C03643=1208.967,92.723,-48.603,-178.715,5.757,148.635
C03644=1208.971,92.474,-48.585,-178.717,5.756,148.636
C03645=1208.975,92.224,-48.566,-178.719,5.755,148.636
C03646=1208.980,91.975,-48.548,-178.723,5.754,148.637
C03647=1208.985,91.726,-48.530,-178.725,5.753,148.637
C03648=1208.990,91.477,-48.512,-178.727,5.752,148.638
C03649=1208.996,91.227,-48.494,-178.731,5.751,148.639
C03650=1209.000,90.977,-48.475,-178.733,5.750,148.639
C03651=1209.005,90.728,-48.457,-178.735,5.749,148.640
C03652=1209.010,90.479,-48.440,-178.737,5.748,148.640
C03653=1209.015,90.230,-48.422,-178.741,5.747,148.641
C03654=1209.020,89.981,-48.404,-178.743,5.746,148.642
C03655=1209.025,89.732,-48.386,-178.745,5.746,148.642
C03656=1209.029,89.482,-48.367,-178.748,5.745,148.643
C03657=1209.034,89.232,-48.349,-178.751,5.744,148.643
C03658=1209.039,88.983,-48.331,-178.753,5.743,148.644
C03659=1209.044,88.734,-48.313,-178.756,5.742,148.644
C03660=1209.049,88.485,-48.295,-178.758,5.741,148.645
C03661=1209.054,88.236,-48.277,-178.761,5.740,148.645
C03662=1209.059,87.987,-48.259,-178.764,5.739,148.646
C03663=1209.064,87.736,-48.240,-178.766,5.738,148.646
C03664=1209.068,87.487,-48.222,-178.769,5.738,148.647
C03665=1209.073,87.238,-48.204,-178.771,5.736,148.648
C03666=1209.078,86.989,-48.186,-178.774,5.735,148.648
C03667=1209.083,86.740,-48.168,-178.777,5.735,148.649
C03668=1209.088,86.491,-48.151,-178.779,5.734,148.649
C03669=1209.093,86.241,-48.133,-178.782,5.732,148.650
C03670=1209.097,85.993,-48.115,-178.785,5.732,148.651
C03671=1209.102,85.743,-48.097,-178.787,5.731,148.651
C03672=1209.107,85.493,-48.080,-178.789,5.730,148.652
C03673=1209.112,85.244,-48.062,-178.793,5.729,148.652
C03674=1209.117,84.994,-48.044,-178.795,5.728,148.653
C03675=1209.121,84.745,-48.026,-178.797,5.727,148.653
C03676=1209.126,84.496,-48.008,-178.799,5.726,148.654
C03677=1209.131,84.247,-47.990,-178.803,5.725,148.654
C03678=1209.137,83.997,-47.972,-178.805,5.725,148.655
C03679=1209.141,83.748,-47.954,-178.807,5.724,148.655
C03680=1209.146,83.499,-47.936,-178.810,5.723,148.656
C03681=1209.151,83.250,-47.918,-178.813,5.722,148.657
C03682=1209.156,83.000,-47.900,-178.815,5.721,148.657
C03683=1209.161,82.751,-47.883,-178.818,5.720,148.658
C03684=1209.166,82.501,-47.865,-178.821,5.720,148.659
C03685=1209.170,82.253,-47.848,-178.823,5.719,148.659
C03686=1209.175,82.003,-47.829,-178.826,5.717,148.660
C03687=1209.180,81.753,-47.812,-178.829,5.717,148.660
C03688=1209.186,81.485,-47.793,-178.831,5.716,148.661
C03689=1209.191,81.217,-47.774,-178.834,5.714,148.661
C03690=1209.196,80.948,-47.755,-178.837,5.714,148.662
C03691=1209.201,80.680,-47.736,-178.839,5.713,148.663
C03692=1209.206,80.431,-47.718,-178.842,5.712,148.663
C03693=1209.211,80.181,-47.700,-178.844,5.711,148.664
C03694=1209.216,79.932,-47.682,-178.847,5.710,148.664
C03695=1209.220,79.683,-47.665,-178.850,5.710,148.665
C03696=1209.226,79.433,-47.648,-178.852,5.709,148.665
C03697=1209.231,79.184,-47.630,-178.855,5.707,148.666
C03698=1209.236,78.935,-47.612,-178.858,5.707,148.667
C03699=1209.241,78.685,-47.595,-178.860,5.706,148.667
C03700=1209.245,78.436,-47.577,-178.862,5.705,148.668
C03701=1209.250,78.186,-47.560,-178.865,5.705,148.669
C03702=1209.255,77.937,-47.542,-178.868,5.703,148.669
C03703=1209.260,77.688,-47.524,-178.870,5.702,148.670
C03704=1209.264,77.439,-47.507,-178.873,5.702,148.670
C03705=1209.269,77.189,-47.489,-178.875,5.701,148.671
C03706=1209.275,76.940,-47.472,-178.878,5.700,148.671
C03707=1209.279,76.690,-47.454,-178.881,5.699,148.672
C03708=1209.284,76.441,-47.437,-178.883,5.698,148.672
C03709=1209.289,76.192,-47.419,-178.886,5.698,148.673
C03710=1209.294,75.942,-47.402,-178.888,5.697,148.674
C03711=1209.300,75.693,-47.385,-178.891,5.696,148.674
C03712=1209.304,75.444,-47.368,-178.894,5.695,148.675
C03713=1209.309,75.195,-47.350,-178.896,5.694,148.675
C03714=1209.314,74.945,-47.333,-178.898,5.693,148.676
C03715=1209.318,74.696,-47.315,-178.901,5.693,148.677
C03716=1209.324,74.446,-47.298,-178.904,5.692,148.677
C03717=1209.329,74.197,-47.280,-178.906,5.691,148.678
C03718=1209.334,73.947,-47.263,-178.909,5.690,148.678
C03719=1209.338,73.699,-47.245,-178.912,5.689,148.679
C03720=1209.343,73.449,-47.228,-178.914,5.688,148.679
C03721=1209.348,73.200,-47.210,-178.916,5.688,148.680
C03722=1209.353,72.950,-47.193,-178.919,5.687,148.681
C03723=1209.358,72.701,-47.177,-178.922,5.685,148.681
C03724=1209.362,72.452,-47.159,-178.924,5.685,148.682
C03725=1209.368,72.202,-47.142,-178.927,5.684,148.682
C03726=1209.373,71.953,-47.124,-178.930,5.684,148.683
C03727=1209.377,71.704,-47.107,-178.932,5.683,148.684
C03728=1209.382,71.454,-47.090,-178.934,5.682,148.684
C03729=1209.387,71.205,-47.072,-178.937,5.682,148.685
C03730=1209.392,70.956,-47.056,-178.940,5.680,148.685
C03731=1209.398,70.706,-47.038,-178.942,5.679,148.686
C03732=1209.402,70.457,-47.021,-178.945,5.679,148.687
C03733=1209.407,70.207,-47.004,-178.947,5.678,148.687
C03734=1209.412,69.958,-46.987,-178.950,5.677,148.688
C03735=1209.416,69.709,-46.969,-178.952,5.677,148.688
C03736=1209.422,69.459,-46.952,-178.956,5.675,148.689
C03737=1209.427,69.210,-46.936,-178.958,5.674,148.689
C03738=1209.432,68.961,-46.918,-178.960,5.674,148.690
C03739=1209.436,68.712,-46.901,-178.963,5.673,148.691
C03740=1209.441,68.462,-46.884,-178.965,5.672,148.691
C03741=1209.446,68.212,-46.867,-178.968,5.672,148.692
C03742=1209.451,67.963,-46.849,-178.970,5.671,148.693
C03743=1209.456,67.714,-46.833,-178.973,5.669,148.693
C03744=1209.461,67.465,-46.815,-178.976,5.669,148.694
C03745=1209.465,67.215,-46.799,-178.978,5.668,148.694
C03746=1209.470,66.966,-46.781,-178.981,5.668,148.695
C03747=1209.475,66.716,-46.764,-178.983,5.667,148.695
C03748=1209.481,66.467,-46.747,-178.986,5.666,148.696
C03749=1209.485,66.218,-46.731,-178.988,5.666,148.697
C03750=1209.490,65.968,-46.713,-178.991,5.664,148.697
C03751=1209.495,65.719,-46.697,-178.994,5.663,148.698
C03752=1209.500,65.470,-46.679,-178.996,5.663,148.698
C03753=1209.505,65.221,-46.662,-178.999,5.662,148.699
C03754=1209.510,64.971,-46.645,-179.001,5.661,148.700
C03755=1209.514,64.721,-46.628,-179.004,5.661,148.700
C03756=1209.520,64.471,-46.611,-179.007,5.660,148.701
C03757=1209.525,64.223,-46.595,-179.009,5.659,148.701
C03758=1209.529,63.973,-46.578,-179.012,5.658,148.702
C03759=1209.534,63.723,-46.561,-179.014,5.657,148.703
C03760=1209.539,63.475,-46.544,-179.017,5.657,148.703
C03761=1209.544,63.225,-46.527,-179.019,5.656,148.704
C03762=1209.549,62.976,-46.510,-179.022,5.655,148.704
C03763=1209.554,62.726,-46.493,-179.025,5.655,148.705
C03764=1209.559,62.477,-46.476,-179.027,5.654,148.706
C03765=1209.564,62.228,-46.460,-179.029,5.653,148.706
C03766=1209.569,61.978,-46.442,-179.033,5.652,148.707
C03767=1209.573,61.729,-46.426,-179.035,5.651,148.707
C03768=1209.579,61.480,-46.409,-179.037,5.651,148.708
C03769=1209.584,61.230,-46.392,-179.040,5.650,148.709
C03770=1209.588,60.981,-46.376,-179.043,5.649,148.709
C03771=1209.594,60.732,-46.359,-179.045,5.649,148.710
C03772=1209.599,60.482,-46.342,-179.047,5.648,148.710
C03773=1209.603,60.233,-46.325,-179.050,5.647,148.711
C03774=1209.609,59.983,-46.308,-179.053,5.647,148.712
C03775=1209.613,59.734,-46.292,-179.055,5.646,148.712
C03776=1209.618,59.484,-46.275,-179.058,5.645,148.713
C03777=1209.623,59.235,-46.258,-179.061,5.644,148.713
C03778=1209.628,58.986,-46.241,-179.063,5.643,148.714
C03779=1209.633,58.736,-46.226,-179.066,5.643,148.715
C03780=1209.637,58.486,-46.209,-179.068,5.642,148.715
C03781=1209.643,58.237,-46.192,-179.071,5.641,148.716
C03782=1209.648,57.988,-46.175,-179.073,5.641,148.717
C03783=1209.653,57.739,-46.159,-179.076,5.640,148.717
C03784=1209.658,57.489,-46.142,-179.078,5.639,148.718
C03785=1209.662,57.240,-46.125,-179.081,5.639,148.718
C03786=1209.667,56.991,-46.109,-179.084,5.638,148.719
C03787=1209.672,56.741,-46.092,-179.087,5.637,148.720
C03788=1209.677,56.491,-46.076,-179.089,5.636,148.720
C03789=1209.683,56.242,-46.059,-179.091,5.636,148.721
C03790=1209.687,55.993,-46.043,-179.094,5.635,148.721
C03791=1209.692,55.743,-46.026,-179.097,5.634,148.722
C03792=1209.698,55.474,-46.008,-179.099,5.634,148.723
C03793=1209.703,55.207,-45.991,-179.102,5.633,148.723
C03794=1209.708,54.938,-45.972,-179.105,5.632,148.724
C03795=1209.713,54.670,-45.955,-179.107,5.631,148.724
C03796=1209.719,54.420,-45.938,-179.110,5.630,148.725
C03797=1209.724,54.171,-45.922,-179.112,5.630,148.726
C03798=1209.728,53.921,-45.905,-179.115,5.629,148.726
C03799=1209.733,53.671,-45.889,-179.118,5.629,148.727
C03800=1209.738,53.423,-45.873,-179.120,5.628,148.728
C03801=1209.743,53.173,-45.856,-179.123,5.627,148.728
C03802=1209.749,52.923,-45.840,-179.125,5.627,148.729
C03803=1209.753,52.674,-45.823,-179.128,5.626,148.730
C03804=1209.758,52.425,-45.807,-179.130,5.625,148.730
C03805=1209.763,52.176,-45.790,-179.133,5.624,148.731
C03806=1209.767,51.926,-45.774,-179.136,5.623,148.731
C03807=1209.772,51.677,-45.758,-179.138,5.623,148.732
C03808=1209.778,51.427,-45.741,-179.141,5.622,148.732
C03809=1209.783,51.178,-45.725,-179.143,5.621,148.733
C03810=1209.788,50.928,-45.709,-179.146,5.621,148.734
C03811=1209.793,50.679,-45.692,-179.148,5.620,148.734
C03812=1209.797,50.429,-45.676,-179.151,5.619,148.735
C03813=1209.802,50.180,-45.660,-179.153,5.619,148.736
C03814=1209.807,49.930,-45.644,-179.156,5.618,148.736
C03815=1209.812,49.682,-45.628,-179.159,5.618,148.737
C03816=1209.817,49.432,-45.611,-179.161,5.617,148.738
C03817=1209.822,49.183,-45.596,-179.163,5.616,148.738
C03818=1209.827,48.933,-45.579,-179.166,5.616,148.739
C03819=1209.833,48.683,-45.563,-179.169,5.615,148.739
C03820=1209.837,48.434,-45.546,-179.171,5.615,148.740
C03821=1209.843,48.185,-45.530,-179.173,5.614,148.740
C03822=1209.847,47.935,-45.514,-179.176,5.613,148.741
C03823=1209.852,47.686,-45.498,-179.179,5.613,148.742
C03824=1209.857,47.436,-45.482,-179.181,5.612,148.743
C03825=1209.862,47.187,-45.465,-179.185,5.611,148.743
C03826=1209.867,46.937,-45.449,-179.187,5.610,148.744
C03827=1209.872,46.689,-45.433,-179.189,5.609,148.744
C03828=1209.877,46.438,-45.417,-179.192,5.609,148.745
C03829=1209.882,46.190,-45.401,-179.195,5.608,148.746
C03830=1209.887,45.940,-45.385,-179.197,5.608,148.746
C03831=1209.892,45.691,-45.368,-179.199,5.607,148.747
C03832=1209.896,45.441,-45.353,-179.202,5.606,148.747
C03833=1209.902,45.191,-45.337,-179.205,5.606,148.748
C03834=1209.906,44.942,-45.320,-179.207,5.605,148.749
C03835=1209.912,44.692,-45.305,-179.210,5.605,148.749
C03836=1209.916,44.443,-45.288,-179.212,5.604,148.750
C03837=1209.922,44.193,-45.272,-179.215,5.603,148.751
C03838=1209.927,43.945,-45.256,-179.217,5.603,148.751
C03839=1209.931,43.695,-45.241,-179.220,5.602,148.752
C03840=1209.936,43.445,-45.225,-179.222,5.601,148.752
C03841=1209.941,43.196,-45.209,-179.225,5.601,148.753
C03842=1209.946,42.947,-45.193,-179.227,5.600,148.754
C03843=1209.951,42.696,-45.177,-179.230,5.600,148.754
C03844=1209.956,42.448,-45.161,-179.233,5.599,148.755
C03845=1209.961,42.198,-45.145,-179.235,5.598,148.755
C03846=1209.966,41.949,-45.128,-179.237,5.598,148.756
C03847=1209.971,41.699,-45.113,-179.240,5.597,148.757
C03848=1209.976,41.449,-45.097,-179.243,5.597,148.757
C03849=1209.981,41.200,-45.081,-179.245,5.596,148.758
C03850=1209.986,40.951,-45.066,-179.248,5.595,148.759
C03851=1209.990,40.701,-45.050,-179.250,5.595,148.759
C03852=1209.996,40.452,-45.034,-179.253,5.594,148.760
C03853=1210.001,40.203,-45.018,-179.255,5.594,148.761
C03854=1210.006,39.953,-45.002,-179.258,5.593,148.761
C03855=1210.011,39.704,-44.986,-179.260,5.592,148.762
C03856=1210.016,39.454,-44.970,-179.263,5.592,148.762
C03857=1210.020,39.205,-44.955,-179.266,5.591,148.763
C03858=1210.026,38.956,-44.939,-179.268,5.590,148.764
C03859=1210.030,38.706,-44.923,-179.271,5.590,148.764
C03860=1210.036,38.456,-44.907,-179.273,5.589,148.765
C03861=1210.041,38.207,-44.891,-179.276,5.588,148.766
C03862=1210.046,37.957,-44.875,-179.278,5.588,148.766
C03863=1210.050,37.708,-44.860,-179.281,5.587,148.767
C03864=1210.056,37.459,-44.845,-179.284,5.587,148.768
C03865=1210.060,37.209,-44.829,-179.286,5.586,148.768
C03866=1210.066,36.960,-44.812,-179.288,5.585,148.769
C03867=1210.071,36.710,-44.797,-179.291,5.585,148.769
C03868=1210.075,36.461,-44.781,-179.294,5.584,148.770
C03869=1210.080,36.211,-44.766,-179.296,5.584,148.771
C03870=1210.086,35.962,-44.750,-179.299,5.583,148.771
C03871=1210.091,35.712,-44.735,-179.301,5.582,148.772
C03872=1210.095,35.463,-44.719,-179.304,5.582,148.773
C03873=1210.101,35.213,-44.704,-179.306,5.581,148.773
C03874=1210.106,34.965,-44.687,-179.309,5.581,148.774
C03875=1210.110,34.714,-44.671,-179.312,5.580,148.775
C03876=1210.115,34.465,-44.656,-179.314,5.580,148.775
C03877=1210.120,34.216,-44.641,-179.316,5.579,148.776
C03878=1210.125,33.966,-44.625,-179.319,5.578,148.776
C03879=1210.130,33.717,-44.610,-179.322,5.578,148.777
C03880=1210.135,33.467,-44.594,-179.324,5.577,148.778
C03881=1210.141,33.218,-44.579,-179.327,5.577,148.778
C03882=1210.145,32.968,-44.563,-179.330,5.576,148.779
C03883=1210.150,32.719,-44.548,-179.332,5.575,148.779
C03884=1210.155,32.469,-44.532,-179.334,5.575,148.780
C03885=1210.161,32.220,-44.517,-179.336,5.575,148.781
C03886=1210.165,31.970,-44.501,-179.339,5.574,148.782
C03887=1210.170,31.721,-44.486,-179.342,5.574,148.782
C03888=1210.175,31.472,-44.471,-179.344,5.573,148.783
C03889=1210.180,31.222,-44.455,-179.347,5.573,148.783
C03890=1210.185,30.972,-44.439,-179.349,5.572,148.784
C03891=1210.190,30.723,-44.424,-179.352,5.571,148.785
C03892=1210.195,30.474,-44.408,-179.355,5.571,148.785
C03893=1210.201,30.224,-44.393,-179.357,5.570,148.786
C03894=1210.205,29.975,-44.378,-179.360,5.570,148.787
C03895=1210.210,29.725,-44.362,-179.362,5.569,148.787
C03896=1210.216,29.456,-44.346,-179.365,5.568,148.788
C03897=1210.221,29.188,-44.329,-179.367,5.568,148.789
C03898=1210.226,28.919,-44.312,-179.370,5.568,148.789
C03899=1210.232,28.650,-44.296,-179.373,5.567,148.790
C03900=1210.237,28.401,-44.281,-179.375,5.566,148.791
C03901=1210.242,28.152,-44.265,-179.378,5.566,148.791
C03902=1210.246,27.902,-44.250,-179.380,5.565,148.792
C03903=1210.252,27.652,-44.234,-179.383,5.565,148.793
C03904=1210.256,27.403,-44.219,-179.386,5.564,148.793
C03905=1210.262,27.153,-44.205,-179.388,5.564,148.794
C03906=1210.267,26.904,-44.190,-179.391,5.563,148.794
C03907=1210.272,26.655,-44.174,-179.393,5.562,148.795
C03908=1210.277,26.405,-44.158,-179.396,5.562,148.796
C03909=1210.281,26.156,-44.143,-179.398,5.561,148.796
C03910=1210.287,25.906,-44.128,-179.401,5.561,148.797
C03911=1210.292,25.657,-44.113,-179.404,5.560,148.798
C03912=1210.297,25.407,-44.098,-179.406,5.560,148.798
C03913=1210.302,25.158,-44.083,-179.409,5.559,148.799
C03914=1210.307,24.908,-44.067,-179.411,5.559,148.800
C03915=1210.311,24.658,-44.052,-179.413,5.559,148.800
C03916=1210.317,24.409,-44.037,-179.416,5.558,148.801
C03917=1210.322,24.160,-44.022,-179.419,5.557,148.802
C03918=1210.327,23.910,-44.006,-179.421,5.557,148.802
C03919=1210.332,23.661,-43.992,-179.423,5.556,148.803
C03920=1210.337,23.412,-43.977,-179.426,5.556,148.803
C03921=1210.342,23.162,-43.961,-179.429,5.555,148.804
C03922=1210.346,22.912,-43.947,-179.431,5.555,148.805
C03923=1210.352,22.662,-43.931,-179.434,5.554,148.805
C03924=1210.356,22.413,-43.916,-179.437,5.553,148.806
C03925=1210.362,22.164,-43.900,-179.439,5.553,148.807
C03926=1210.367,21.914,-43.886,-179.441,5.552,148.807
C03927=1210.372,21.665,-43.871,-179.443,5.552,148.808
C03928=1210.377,21.416,-43.856,-179.446,5.552,148.809
C03929=1210.382,21.166,-43.841,-179.449,5.551,148.809
C03930=1210.387,20.917,-43.826,-179.451,5.551,148.810
C03931=1210.392,20.667,-43.811,-179.454,5.550,148.811
C03932=1210.397,20.417,-43.796,-179.457,5.550,148.811
C03933=1210.401,20.168,-43.781,-179.459,5.549,148.812
C03934=1210.406,19.918,-43.766,-179.462,5.548,148.813
C03935=1210.412,19.669,-43.751,-179.464,5.548,148.813
C03936=1210.417,19.419,-43.736,-179.467,5.547,148.814
C03937=1210.422,19.169,-43.721,-179.469,5.547,148.815
C03938=1210.427,18.920,-43.706,-179.472,5.547,148.815
C03939=1210.432,18.671,-43.692,-179.474,5.547,148.816
C03940=1210.437,18.421,-43.676,-179.476,5.546,148.816
C03941=1210.442,18.171,-43.662,-179.479,5.545,148.817
C03942=1210.447,17.922,-43.647,-179.482,5.545,148.818
C03943=1210.452,17.672,-43.632,-179.484,5.544,148.818
C03944=1210.457,17.423,-43.617,-179.487,5.544,148.819
C03945=1210.462,17.174,-43.603,-179.490,5.543,148.820
C03946=1210.467,16.924,-43.587,-179.492,5.543,148.820
C03947=1210.472,16.674,-43.573,-179.494,5.542,148.821
C03948=1210.477,16.425,-43.558,-179.496,5.542,148.822
C03949=1210.482,16.176,-43.543,-179.499,5.541,148.822
C03950=1210.487,15.926,-43.528,-179.502,5.541,148.823
C03951=1210.492,15.677,-43.514,-179.504,5.540,148.824
C03952=1210.497,15.427,-43.499,-179.507,5.540,148.824
C03953=1210.503,15.177,-43.484,-179.510,5.539,148.825
C03954=1210.507,14.928,-43.469,-179.512,5.539,148.826
C03955=1210.512,14.679,-43.454,-179.515,5.538,148.826
C03956=1210.517,14.430,-43.439,-179.517,5.538,148.827
C03957=1210.523,14.180,-43.425,-179.519,5.538,148.828
C03958=1210.528,13.930,-43.410,-179.522,5.537,148.828
C03959=1210.532,13.681,-43.395,-179.525,5.537,148.829
C03960=1210.537,13.431,-43.381,-179.527,5.536,148.830
C03961=1210.542,13.182,-43.365,-179.530,5.536,148.830
C03962=1210.547,12.932,-43.351,-179.532,5.535,148.831
C03963=1210.552,12.682,-43.337,-179.535,5.534,148.831
C03964=1210.557,12.433,-43.322,-179.537,5.535,148.832
C03965=1210.562,12.183,-43.308,-179.539,5.534,148.833
C03966=1210.568,11.933,-43.293,-179.542,5.534,148.833
C03967=1210.572,11.684,-43.278,-179.545,5.533,148.834
C03968=1210.577,11.435,-43.263,-179.547,5.532,148.835
C03969=1210.582,11.185,-43.249,-179.550,5.532,148.836
C03970=1210.588,10.936,-43.235,-179.552,5.531,148.836
C03971=1210.593,10.686,-43.220,-179.555,5.531,148.837
C03972=1210.598,10.437,-43.205,-179.557,5.531,148.837
C03973=1210.603,10.188,-43.190,-179.559,5.530,148.838
C03974=1210.608,9.938,-43.176,-179.562,5.530,148.839
C03975=1210.613,9.688,-43.162,-179.565,5.529,148.839
C03976=1210.618,9.439,-43.148,-179.567,5.529,148.840
C03977=1210.623,9.189,-43.132,-179.570,5.528,148.841
C03978=1210.628,8.939,-43.118,-179.573,5.528,148.841
C03979=1210.633,8.690,-43.103,-179.574,5.528,148.842
C03980=1210.638,8.440,-43.089,-179.577,5.527,148.843
C03981=1210.643,8.192,-43.075,-179.580,5.527,148.843
C03982=1210.648,7.942,-43.060,-179.582,5.526,148.844
C03983=1210.653,7.692,-43.046,-179.585,5.526,148.845
C03984=1210.658,7.442,-43.032,-179.588,5.525,148.845
C03985=1210.663,7.193,-43.017,-179.590,5.525,148.846
C03986=1210.668,6.943,-43.002,-179.592,5.525,148.847
C03987=1210.673,6.694,-42.988,-179.594,5.524,148.847
C03988=1210.678,6.444,-42.973,-179.597,5.524,148.848
C03989=1210.684,6.195,-42.959,-179.600,5.523,148.849
C03990=1210.689,5.945,-42.945,-179.602,5.523,148.849
C03991=1210.694,5.695,-42.931,-179.605,5.522,148.850
C03992=1210.698,5.446,-42.916,-179.607,5.522,148.851
C03993=1210.703,5.197,-42.902,-179.610,5.522,148.851
C03994=1210.708,4.947,-42.887,-179.612,5.521,148.852
C03995=1210.713,4.697,-42.873,-179.615,5.521,148.853
C03996=1210.719,4.448,-42.859,-179.617,5.520,148.853
C03997=1210.724,4.199,-42.845,-179.620,5.519,148.854
C03998=1210.729,3.949,-42.831,-179.623,5.519,148.855
C03999=1210.734,3.699,-42.816,-179.625,5.519,148.855
C04000=1210.739,3.430,-42.801,-179.627,5.519,148.856
C04001=1210.744,3.161,-42.786,-179.630,5.518,148.857
C04002=1210.750,2.893,-42.770,-179.633,5.518,148.857
C04003=1210.756,2.623,-42.755,-179.636,5.518,148.858
C04004=1210.761,2.373,-42.740,-179.638,5.517,148.859
C04005=1210.766,2.124,-42.726,-179.641,5.516,148.859
C04006=1210.771,1.874,-42.712,-179.643,5.516,148.860
C04007=1210.776,1.625,-42.698,-179.646,5.515,148.861
C04008=1210.781,1.376,-42.684,-179.648,5.516,148.861
C04009=1210.786,1.126,-42.670,-179.651,5.515,148.862
C04010=1210.791,0.876,-42.656,-179.653,5.514,148.863
C04011=1210.796,0.626,-42.641,-179.656,5.514,148.863
C04012=1210.801,0.377,-42.627,-179.659,5.513,148.864
C04013=1210.806,0.128,-42.613,-179.661,5.513,148.865
C04014=1210.811,-0.122,-42.599,-179.663,5.513,148.865
C04015=1210.816,-0.372,-42.585,-179.665,5.512,148.866
C04016=1210.822,-0.621,-42.571,-179.668,5.512,148.867
C04017=1210.827,-0.870,-42.556,-179.671,5.511,148.867
C04018=1210.832,-1.120,-42.542,-179.673,5.511,148.868
C04019=1210.836,-1.370,-42.528,-179.675,5.511,148.869
C04020=1210.842,-1.619,-42.514,-179.678,5.511,148.869
C04021=1210.846,-1.868,-42.500,-179.681,5.510,148.870
C04022=1210.851,-2.118,-42.486,-179.683,5.510,148.871
C04023=1210.856,-2.368,-42.472,-179.686,5.509,148.871
C04024=1210.862,-2.617,-42.458,-179.688,5.509,148.872
C04025=1210.867,-2.867,-42.444,-179.690,5.509,148.873
C04026=1210.872,-3.117,-42.430,-179.693,5.508,148.873
C04027=1210.877,-3.366,-42.416,-179.696,5.508,148.874
C04028=1210.882,-3.615,-42.402,-179.698,5.507,148.875
C04029=1210.887,-3.865,-42.388,-179.700,5.507,148.875
C04030=1210.892,-4.115,-42.374,-179.703,5.507,148.876
C04031=1210.897,-4.364,-42.361,-179.706,5.506,148.877
C04032=1210.902,-4.614,-42.346,-179.708,5.506,148.877
C04033=1210.907,-4.864,-42.332,-179.711,5.505,148.878
C04034=1210.913,-5.113,-42.318,-179.713,5.505,148.879
C04035=1210.917,-5.362,-42.304,-179.715,5.505,148.879
C04036=1210.922,-5.612,-42.290,-179.718,5.504,148.880
C04037=1210.927,-5.862,-42.277,-179.721,5.504,148.881
C04038=1210.933,-6.111,-42.263,-179.723,5.503,148.881
C04039=1210.938,-6.361,-42.248,-179.725,5.504,148.882
C04040=1210.942,-6.610,-42.235,-179.728,5.503,148.883
C04041=1210.948,-6.860,-42.222,-179.731,5.503,148.883
C04042=1210.953,-7.110,-42.207,-179.733,5.502,148.884
C04043=1210.958,-7.359,-42.193,-179.735,5.501,148.885
C04044=1210.963,-7.608,-42.180,-179.737,5.502,148.885
C04045=1210.968,-7.858,-42.166,-179.740,5.501,148.886
C04046=1210.973,-8.108,-42.152,-179.743,5.501,148.887
C04047=1210.978,-8.357,-42.138,-179.745,5.500,148.887
C04048=1210.983,-8.607,-42.125,-179.748,5.500,148.888
C04049=1210.989,-8.856,-42.111,-179.750,5.500,148.889
C04050=1210.994,-9.106,-42.097,-179.753,5.499,148.889
C04051=1210.999,-9.356,-42.083,-179.755,5.499,148.890
C04052=1211.004,-9.605,-42.070,-179.758,5.498,148.891
C04053=1211.009,-9.854,-42.056,-179.760,5.498,148.891
C04054=1211.014,-10.105,-42.042,-179.762,5.498,148.892
C04055=1211.019,-10.353,-42.029,-179.765,5.497,148.893
C04056=1211.024,-10.603,-42.014,-179.768,5.497,148.893
C04057=1211.029,-10.854,-42.001,-179.770,5.496,148.894
C04058=1211.034,-11.102,-41.988,-179.772,5.497,148.895
C04059=1211.039,-11.352,-41.973,-179.775,5.496,148.895
C04060=1211.044,-11.602,-41.960,-179.778,5.496,148.896
C04061=1211.049,-11.851,-41.946,-179.780,5.495,148.897
C04062=1211.054,-12.101,-41.933,-179.782,5.496,148.898
C04063=1211.060,-12.350,-41.919,-179.785,5.495,148.898
C04064=1211.064,-12.600,-41.906,-179.787,5.494,148.899
C04065=1211.070,-12.849,-41.892,-179.790,5.494,148.899
C04066=1211.075,-13.099,-41.878,-179.793,5.493,148.900
C04067=1211.080,-13.348,-41.865,-179.795,5.494,148.901
C04068=1211.085,-13.598,-41.851,-179.797,5.493,148.901
C04069=1211.090,-13.848,-41.837,-179.800,5.493,148.902
C04070=1211.095,-14.097,-41.824,-179.803,5.492,148.903
C04071=1211.100,-14.347,-41.811,-179.805,5.492,148.904
C04072=1211.105,-14.596,-41.797,-179.807,5.492,148.904
C04073=1211.110,-14.846,-41.784,-179.810,5.491,148.905
C04074=1211.116,-15.095,-41.770,-179.813,5.491,148.906
C04075=1211.120,-15.345,-41.757,-179.814,5.491,148.906
C04076=1211.126,-15.594,-41.743,-179.817,5.490,148.907
C04077=1211.130,-15.845,-41.730,-179.820,5.490,148.907
C04078=1211.136,-16.094,-41.716,-179.822,5.489,148.908
C04079=1211.141,-16.344,-41.702,-179.824,5.490,148.909
C04080=1211.145,-16.593,-41.689,-179.827,5.489,148.910
C04081=1211.151,-16.843,-41.676,-179.830,5.489,148.910
C04082=1211.156,-17.093,-41.663,-179.832,5.488,148.911
C04083=1211.161,-17.342,-41.649,-179.834,5.489,148.912
C04084=1211.166,-17.592,-41.636,-179.837,5.488,148.912
C04085=1211.171,-17.841,-41.622,-179.840,5.488,148.913
C04086=1211.176,-18.091,-41.609,-179.842,5.487,148.914
C04087=1211.182,-18.341,-41.596,-179.844,5.487,148.914
C04088=1211.186,-18.590,-41.582,-179.847,5.487,148.915
C04089=1211.192,-18.840,-41.569,-179.849,5.486,148.916
C04090=1211.197,-19.089,-41.554,-179.852,5.486,148.916
C04091=1211.202,-19.339,-41.542,-179.854,5.486,148.917
C04092=1211.207,-19.589,-41.528,-179.857,5.485,148.918
C04093=1211.212,-19.838,-41.515,-179.859,5.485,148.918
C04094=1211.218,-20.087,-41.502,-179.862,5.484,148.919
C04095=1211.222,-20.337,-41.489,-179.864,5.485,148.920
C04096=1211.227,-20.586,-41.475,-179.867,5.484,148.920
C04097=1211.232,-20.836,-41.462,-179.869,5.484,148.921
C04098=1211.237,-21.086,-41.449,-179.872,5.483,148.922
C04099=1211.242,-21.335,-41.435,-179.874,5.483,148.922
C04100=1211.248,-21.585,-41.422,-179.876,5.483,148.923
C04101=1211.253,-21.835,-41.409,-179.879,5.482,148.924
C04102=1211.258,-22.084,-41.396,-179.881,5.483,148.924
C04103=1211.263,-22.334,-41.382,-179.884,5.482,148.925
C04104=1211.268,-22.603,-41.369,-179.886,5.482,148.926
C04105=1211.274,-22.873,-41.354,-179.889,5.481,148.926
C04106=1211.280,-23.143,-41.339,-179.892,5.481,148.927
C04107=1211.285,-23.412,-41.326,-179.895,5.481,148.928
C04108=1211.290,-23.661,-41.312,-179.897,5.481,148.929
C04109=1211.295,-23.911,-41.299,-179.899,5.480,148.929
C04110=1211.300,-24.161,-41.286,-179.902,5.479,148.930
C04111=1211.306,-24.410,-41.273,-179.904,5.479,148.931
C04112=1211.310,-24.660,-41.260,-179.906,5.479,148.931
C04113=1211.316,-24.909,-41.246,-179.909,5.479,148.932
C04114=1211.321,-25.159,-41.234,-179.912,5.478,148.933
C04115=1211.325,-25.409,-41.221,-179.914,5.479,148.933
C04116=1211.331,-25.658,-41.207,-179.917,5.478,148.934
C04117=1211.336,-25.908,-41.194,-179.919,5.478,148.935
C04118=1211.341,-26.158,-41.182,-179.922,5.477,148.936
C04119=1211.346,-26.407,-41.168,-179.924,5.478,148.936
C04120=1211.351,-26.657,-41.155,-179.927,5.477,148.937
C04121=1211.356,-26.906,-41.142,-179.929,5.476,148.937
C04122=1211.362,-27.156,-41.129,-179.931,5.477,148.938
C04123=1211.367,-27.406,-41.116,-179.933,5.476,148.939
C04124=1211.372,-27.655,-41.104,-179.936,5.476,148.939
C04125=1211.377,-27.905,-41.090,-179.939,5.475,148.940
C04126=1211.382,-28.155,-41.077,-179.941,5.475,148.941
C04127=1211.387,-28.404,-41.065,-179.944,5.475,148.942
C04128=1211.392,-28.654,-41.051,-179.946,5.474,148.942
C04129=1211.397,-28.903,-41.038,-179.948,5.475,148.943
C04130=1211.402,-29.152,-41.025,-179.951,5.474,148.944
C04131=1211.407,-29.402,-41.012,-179.954,5.474,148.944
C04132=1211.413,-29.652,-40.999,-179.956,5.473,148.945
C04133=1211.418,-29.901,-40.987,-179.958,5.473,148.946
C04134=1211.422,-30.151,-40.974,-179.961,5.473,148.946
C04135=1211.428,-30.401,-40.960,-179.963,5.472,148.947
C04136=1211.433,-30.650,-40.948,-179.965,5.473,148.948
C04137=1211.438,-30.900,-40.935,-179.968,5.472,148.948
C04138=1211.443,-31.149,-40.922,-179.971,5.472,148.949
C04139=1211.449,-31.399,-40.909,-179.973,5.472,148.950
C04140=1211.453,-31.649,-40.896,-179.975,5.472,148.950
C04141=1211.459,-31.898,-40.884,-179.978,5.471,148.951
C04142=1211.464,-32.148,-40.871,-179.981,5.471,148.952
C04143=1211.468,-32.398,-40.858,-179.983,5.471,148.952
C04144=1211.474,-32.647,-40.845,-179.985,5.470,148.953
C04145=1211.479,-32.897,-40.832,-179.988,5.470,148.954
C04146=1211.484,-33.146,-40.820,-179.990,5.470,148.954
C04147=1211.489,-33.396,-40.807,-179.992,5.469,148.955
C04148=1211.495,-33.646,-40.793,-179.995,5.469,148.956
C04149=1211.500,-33.896,-40.782,-179.997,5.469,148.956
C04150=1211.505,-34.146,-40.769,-180.000,5.469,148.957
C04151=1211.510,-34.395,-40.756,179.998,5.468,148.958
C04152=1211.515,-34.644,-40.743,179.996,5.469,148.959
C04153=1211.520,-34.894,-40.731,179.993,5.468,148.959
C04154=1211.525,-35.144,-40.717,179.990,5.468,148.960
C04155=1211.530,-35.393,-40.705,179.988,5.467,148.961
C04156=1211.536,-35.643,-40.692,179.985,5.468,148.961
C04157=1211.541,-35.892,-40.679,179.983,5.467,148.962
C04158=1211.545,-36.142,-40.667,179.981,5.466,148.963
C04159=1211.551,-36.392,-40.655,179.979,5.467,148.963
C04160=1211.556,-36.641,-40.641,179.976,5.466,148.964
C04161=1211.562,-36.891,-40.629,179.973,5.466,148.965
C04162=1211.567,-37.140,-40.616,179.971,5.466,148.965
C04163=1211.571,-37.390,-40.603,179.968,5.466,148.966
C04164=1211.577,-37.640,-40.591,179.966,5.465,148.967
C04165=1211.582,-37.889,-40.579,179.964,5.465,148.967
C04166=1211.587,-38.139,-40.566,179.961,5.465,148.968
C04167=1211.591,-38.389,-40.553,179.958,5.464,148.969
C04168=1211.597,-38.638,-40.541,179.957,5.464,148.969
C04169=1211.603,-38.888,-40.528,179.954,5.464,148.970
C04170=1211.608,-39.138,-40.515,179.951,5.463,148.971
C04171=1211.613,-39.387,-40.503,179.949,5.464,148.971
C04172=1211.617,-39.637,-40.490,179.947,5.463,148.972
C04173=1211.623,-39.887,-40.478,179.944,5.463,148.973
C04174=1211.628,-40.136,-40.465,179.942,5.463,148.973
C04175=1211.633,-40.385,-40.453,179.939,5.463,148.974
C04176=1211.639,-40.635,-40.441,179.937,5.462,148.975
C04177=1211.643,-40.885,-40.428,179.935,5.463,148.976
C04178=1211.648,-41.135,-40.415,179.932,5.462,148.976
C04179=1211.653,-41.384,-40.403,179.929,5.462,148.977
C04180=1211.659,-41.634,-40.391,179.928,5.462,148.977
C04181=1211.664,-41.883,-40.378,179.925,5.461,148.978
C04182=1211.669,-42.133,-40.366,179.922,5.461,148.979
C04183=1211.674,-42.383,-40.353,179.920,5.461,148.980
C04184=1211.679,-42.633,-40.341,179.918,5.461,148.980
C04185=1211.684,-42.882,-40.328,179.915,5.460,148.981
C04186=1211.690,-43.132,-40.316,179.913,5.460,148.982
C04187=1211.695,-43.381,-40.304,179.910,5.460,148.982
C04188=1211.700,-43.630,-40.291,179.908,5.459,148.983
C04189=1211.705,-43.880,-40.279,179.905,5.460,148.984
C04190=1211.710,-44.130,-40.266,179.903,5.459,148.984
C04191=1211.715,-44.380,-40.254,179.900,5.459,148.985
C04192=1211.720,-44.630,-40.242,179.899,5.459,148.986
C04193=1211.725,-44.879,-40.229,179.896,5.458,148.986
C04194=1211.731,-45.129,-40.217,179.893,5.458,148.987
C04195=1211.736,-45.378,-40.205,179.891,5.458,148.988
C04196=1211.741,-45.628,-40.193,179.888,5.458,148.988
C04197=1211.747,-45.877,-40.180,179.886,5.458,148.989
C04198=1211.751,-46.128,-40.168,179.884,5.458,148.990
C04199=1211.756,-46.377,-40.155,179.881,5.457,148.991
C04200=1211.762,-46.627,-40.143,179.879,5.458,148.991
C04201=1211.766,-46.876,-40.131,179.876,5.457,148.992
C04202=1211.771,-47.126,-40.119,179.874,5.457,148.993
C04203=1211.777,-47.376,-40.107,179.872,5.457,148.993
C04204=1211.782,-47.625,-40.094,179.869,5.456,148.994
C04205=1211.787,-47.875,-40.082,179.867,5.456,148.995
C04206=1211.793,-48.124,-40.070,179.865,5.456,148.995
C04207=1211.798,-48.374,-40.058,179.862,5.455,148.996
C04208=1211.803,-48.645,-40.045,179.859,5.455,148.997
C04209=1211.808,-48.914,-40.031,179.857,5.455,148.997
C04210=1211.814,-49.184,-40.019,179.854,5.455,148.998
C04211=1211.820,-49.455,-40.005,179.851,5.455,148.999
C04212=1211.825,-49.704,-39.993,179.849,5.454,149.000
C04213=1211.830,-49.953,-39.981,179.847,5.455,149.000
C04214=1211.835,-50.203,-39.969,179.844,5.454,149.001
C04215=1211.841,-50.453,-39.957,179.842,5.453,149.002
C04216=1211.846,-50.702,-39.944,179.840,5.454,149.002
C04217=1211.851,-50.952,-39.932,179.837,5.453,149.003
C04218=1211.856,-51.202,-39.921,179.835,5.454,149.004
C04219=1211.861,-51.451,-39.908,179.832,5.453,149.004
C04220=1211.866,-51.701,-39.897,179.830,5.453,149.005
C04221=1211.871,-51.950,-39.884,179.828,5.453,149.006
C04222=1211.877,-52.200,-39.872,179.825,5.453,149.006
C04223=1211.882,-52.450,-39.860,179.822,5.452,149.007
C04224=1211.887,-52.699,-39.848,179.821,5.452,149.008
C04225=1211.892,-52.949,-39.836,179.818,5.452,149.008
C04226=1211.898,-53.199,-39.824,179.816,5.452,149.009
C04227=1211.903,-53.448,-39.812,179.813,5.451,149.010
C04228=1211.907,-53.698,-39.800,179.811,5.451,149.010
C04229=1211.913,-53.948,-39.789,179.808,5.451,149.011
C04230=1211.918,-54.197,-39.776,179.806,5.451,149.012
C04231=1211.923,-54.447,-39.764,179.803,5.450,149.013
C04232=1211.928,-54.697,-39.753,179.801,5.451,149.013
C04233=1211.933,-54.946,-39.740,179.798,5.450,149.014
C04234=1211.939,-55.196,-39.728,179.796,5.451,149.015
C04235=1211.944,-55.446,-39.716,179.794,5.450,149.015
C04236=1211.948,-55.695,-39.704,179.791,5.449,149.016
C04237=1211.954,-55.945,-39.693,179.789,5.450,149.017
C04238=1211.959,-56.195,-39.681,179.787,5.449,149.017
C04239=1211.964,-56.444,-39.669,179.784,5.449,149.018
C04240=1211.969,-56.694,-39.657,179.782,5.449,149.019
C04241=1211.975,-56.944,-39.645,179.779,5.449,149.019
C04242=1211.980,-57.194,-39.633,179.777,5.449,149.020
C04243=1211.985,-57.443,-39.622,179.774,5.449,149.021
C04244=1211.990,-57.693,-39.609,179.772,5.448,149.022
C04245=1211.995,-57.942,-39.597,179.770,5.448,149.022
C04246=1212.000,-58.192,-39.586,179.768,5.448,149.023
C04247=1212.005,-58.442,-39.574,179.765,5.448,149.023
C04248=1212.011,-58.692,-39.562,179.763,5.448,149.024
C04249=1212.015,-58.941,-39.550,179.760,5.447,149.025
C04250=1212.021,-59.191,-39.538,179.758,5.447,149.026
C04251=1212.026,-59.441,-39.526,179.755,5.447,149.026
C04252=1212.031,-59.690,-39.515,179.753,5.447,149.027
C04253=1212.037,-59.940,-39.504,179.751,5.447,149.028
C04254=1212.042,-60.190,-39.492,179.748,5.446,149.028
C04255=1212.047,-60.439,-39.480,179.746,5.446,149.029
C04256=1212.052,-60.689,-39.468,179.744,5.446,149.030
C04257=1212.057,-60.938,-39.457,179.742,5.446,149.030
C04258=1212.062,-61.188,-39.445,179.739,5.446,149.031
C04259=1212.068,-61.438,-39.433,179.736,5.445,149.032
C04260=1212.072,-61.688,-39.421,179.734,5.446,149.032
C04261=1212.078,-61.938,-39.410,179.732,5.445,149.033
C04262=1212.082,-62.187,-39.398,179.729,5.446,149.034
C04263=1212.088,-62.437,-39.387,179.727,5.445,149.034
C04264=1212.094,-62.686,-39.374,179.724,5.445,149.035
C04265=1212.098,-62.935,-39.363,179.723,5.445,149.036
C04266=1212.104,-63.185,-39.351,179.720,5.444,149.036
C04267=1212.108,-63.435,-39.340,179.718,5.445,149.037
C04268=1212.114,-63.685,-39.328,179.715,5.444,149.038
C04269=1212.118,-63.935,-39.317,179.712,5.444,149.038
C04270=1212.124,-64.185,-39.305,179.710,5.444,149.039
C04271=1212.130,-64.434,-39.293,179.708,5.444,149.040
C04272=1212.135,-64.683,-39.282,179.706,5.444,149.041
C04273=1212.140,-64.933,-39.270,179.703,5.444,149.041
C04274=1212.145,-65.183,-39.259,179.701,5.443,149.042
C04275=1212.150,-65.433,-39.247,179.699,5.443,149.042
C04276=1212.155,-65.683,-39.235,179.696,5.443,149.043
C04277=1212.161,-65.932,-39.224,179.694,5.443,149.044
C04278=1212.166,-66.181,-39.213,179.691,5.442,149.045
C04279=1212.171,-66.431,-39.201,179.689,5.442,149.045
C04280=1212.176,-66.681,-39.190,179.686,5.442,149.046
C04281=1212.181,-66.931,-39.178,179.684,5.442,149.047
C04282=1212.186,-67.180,-39.166,179.682,5.442,149.047
C04283=1212.192,-67.430,-39.155,179.680,5.441,149.048
C04284=1212.197,-67.679,-39.144,179.677,5.442,149.049
C04285=1212.202,-67.930,-39.132,179.675,5.441,149.049
C04286=1212.207,-68.180,-39.121,179.672,5.441,149.050
C04287=1212.212,-68.429,-39.109,179.670,5.441,149.051
C04288=1212.218,-68.678,-39.098,179.667,5.441,149.051
C04289=1212.223,-68.928,-39.086,179.665,5.441,149.052
C04290=1212.228,-69.178,-39.075,179.663,5.441,149.053
C04291=1212.233,-69.428,-39.063,179.660,5.440,149.054
C04292=1212.239,-69.677,-39.052,179.658,5.440,149.054
C04293=1212.243,-69.926,-39.041,179.656,5.440,149.055
C04294=1212.249,-70.176,-39.029,179.654,5.440,149.055
C04295=1212.254,-70.427,-39.019,179.651,5.440,149.056
C04296=1212.259,-70.677,-39.007,179.649,5.440,149.057
C04297=1212.264,-70.925,-38.996,179.646,5.440,149.058
C04298=1212.270,-71.175,-38.984,179.643,5.439,149.058
C04299=1212.274,-71.425,-38.973,179.641,5.440,149.059
C04300=1212.279,-71.675,-38.961,179.639,5.439,149.059
C04301=1212.286,-71.925,-38.950,179.637,5.439,149.060
C04302=1212.290,-72.174,-38.939,179.634,5.439,149.061
C04303=1212.296,-72.424,-38.927,179.632,5.439,149.062
C04304=1212.300,-72.674,-38.916,179.630,5.439,149.062
C04305=1212.306,-72.923,-38.905,179.627,5.438,149.063
C04306=1212.311,-73.173,-38.894,179.625,5.438,149.064
C04307=1212.316,-73.423,-38.883,179.622,5.438,149.064
C04308=1212.322,-73.672,-38.871,179.620,5.438,149.065
C04309=1212.327,-73.922,-38.860,179.618,5.438,149.066
C04310=1212.332,-74.172,-38.849,179.616,5.438,149.066
C04311=1212.337,-74.422,-38.837,179.613,5.437,149.067
C04312=1212.343,-74.692,-38.826,179.611,5.437,149.068
C04313=1212.348,-74.963,-38.814,179.609,5.437,149.068
C04314=1212.354,-75.233,-38.801,179.606,5.437,149.069
C04315=1212.360,-75.503,-38.789,179.603,5.437,149.070
C04316=1212.365,-75.754,-38.778,179.601,5.437,149.071
C04317=1212.370,-76.004,-38.766,179.598,5.436,149.071
C04318=1212.376,-76.253,-38.756,179.596,5.437,149.072
C04319=1212.380,-76.502,-38.744,179.594,5.436,149.073
C04320=1212.386,-76.753,-38.733,179.591,5.436,149.073
C04321=1212.391,-77.002,-38.722,179.589,5.436,149.074
C04322=1212.396,-77.251,-38.711,179.586,5.436,149.075
C04323=1212.401,-77.502,-38.700,179.584,5.436,149.076
C04324=1212.407,-77.751,-38.689,179.582,5.435,149.076
C04325=1212.412,-78.000,-38.677,179.580,5.436,149.077
C04326=1212.417,-78.251,-38.667,179.577,5.435,149.077
C04327=1212.423,-78.500,-38.655,179.575,5.436,149.078
C04328=1212.428,-78.750,-38.645,179.572,5.435,149.079
C04329=1212.432,-79.000,-38.634,179.570,5.435,149.080
C04330=1212.438,-79.249,-38.623,179.568,5.435,149.080
C04331=1212.443,-79.499,-38.611,179.565,5.434,149.081
C04332=1212.448,-79.749,-38.600,179.563,5.435,149.081
C04333=1212.454,-79.998,-38.590,179.561,5.434,149.082
C04334=1212.458,-80.248,-38.579,179.559,5.435,149.083
C04335=1212.464,-80.497,-38.568,179.556,5.434,149.084
C04336=1212.469,-80.747,-38.557,179.554,5.435,149.084
C04337=1212.474,-80.997,-38.545,179.551,5.434,149.085
C04338=1212.480,-81.247,-38.535,179.549,5.434,149.086
C04339=1212.484,-81.496,-38.524,179.547,5.434,149.086
C04340=1212.490,-81.747,-38.513,179.544,5.433,149.087
C04341=1212.495,-81.996,-38.502,179.542,5.434,149.088
C04342=1212.500,-82.246,-38.491,179.539,5.433,149.088
C04343=1212.506,-82.495,-38.480,179.537,5.433,149.089
C04344=1212.511,-82.745,-38.470,179.535,5.433,149.090
C04345=1212.515,-82.995,-38.458,179.533,5.433,149.090
C04346=1212.522,-83.245,-38.448,179.530,5.433,149.091
C04347=1212.526,-83.494,-38.436,179.528,5.433,149.092
C04348=1212.532,-83.744,-38.426,179.526,5.433,149.092
C04349=1212.537,-83.993,-38.415,179.524,5.433,149.093
C04350=1212.542,-84.244,-38.404,179.521,5.432,149.094
C04351=1212.547,-84.493,-38.393,179.519,5.433,149.094
C04352=1212.552,-84.743,-38.383,179.517,5.432,149.095
C04353=1212.558,-84.992,-38.371,179.514,5.432,149.096
C04354=1212.563,-85.242,-38.361,179.512,5.432,149.096
C04355=1212.568,-85.492,-38.349,179.509,5.431,149.097
C04356=1212.573,-85.742,-38.339,179.507,5.432,149.098
C04357=1212.578,-85.991,-38.328,179.504,5.431,149.099
C04358=1212.584,-86.241,-38.318,179.502,5.432,149.099
C04359=1212.589,-86.491,-38.307,179.500,5.431,149.100
C04360=1212.594,-86.740,-38.296,179.498,5.431,149.100
C04361=1212.600,-86.990,-38.285,179.495,5.431,149.101
C04362=1212.605,-87.239,-38.274,179.493,5.431,149.102
C04363=1212.610,-87.490,-38.263,179.491,5.431,149.103
C04364=1212.615,-87.740,-38.253,179.489,5.431,149.103
C04365=1212.620,-87.989,-38.242,179.486,5.431,149.104
C04366=1212.625,-88.239,-38.231,179.484,5.431,149.104
C04367=1212.631,-88.489,-38.221,179.482,5.430,149.105
C04368=1212.636,-88.738,-38.210,179.479,5.430,149.106
C04369=1212.641,-88.988,-38.200,179.477,5.430,149.107
C04370=1212.646,-89.238,-38.189,179.474,5.430,149.107
C04371=1212.651,-89.487,-38.178,179.472,5.430,149.108
C04372=1212.656,-89.737,-38.168,179.470,5.429,149.108
C04373=1212.662,-89.987,-38.157,179.468,5.430,149.109
C04374=1212.667,-90.236,-38.146,179.465,5.429,149.110
C04375=1212.672,-90.486,-38.136,179.463,5.430,149.111
C04376=1212.677,-90.736,-38.125,179.460,5.429,149.111
C04377=1212.683,-90.985,-38.114,179.458,5.430,149.112
C04378=1212.688,-91.235,-38.104,179.456,5.429,149.113
C04379=1212.693,-91.485,-38.094,179.454,5.429,149.113
C04380=1212.698,-91.735,-38.083,179.451,5.429,149.114
C04381=1212.703,-91.984,-38.072,179.449,5.429,149.115
C04382=1212.708,-92.234,-38.061,179.447,5.429,149.115
C04383=1212.714,-92.484,-38.051,179.445,5.429,149.116
C04384=1212.719,-92.734,-38.041,179.442,5.428,149.117
C04385=1212.724,-92.983,-38.030,179.440,5.429,149.117
C04386=1212.729,-93.233,-38.019,179.438,5.428,149.118
C04387=1212.735,-93.483,-38.009,179.436,5.429,149.119
C04388=1212.741,-93.732,-37.999,179.433,5.428,149.119
C04389=1212.746,-93.982,-37.988,179.430,5.428,149.120
C04390=1212.751,-94.231,-37.977,179.429,5.428,149.121
C04391=1212.756,-94.482,-37.967,179.426,5.427,149.121
C04392=1212.761,-94.731,-37.956,179.424,5.428,149.122
C04393=1212.766,-94.981,-37.946,179.421,5.427,149.123
C04394=1212.772,-95.231,-37.936,179.419,5.428,149.123
C04395=1212.777,-95.481,-37.924,179.416,5.427,149.124
C04396=1212.782,-95.730,-37.914,179.415,5.427,149.125
C04397=1212.788,-95.980,-37.904,179.412,5.427,149.125
C04398=1212.793,-96.230,-37.893,179.410,5.427,149.126
C04399=1212.799,-96.479,-37.883,179.407,5.427,149.127
C04400=1212.803,-96.729,-37.873,179.405,5.427,149.127
C04401=1212.808,-96.979,-37.863,179.403,5.426,149.128
C04402=1212.813,-97.229,-37.852,179.401,5.427,149.129
C04403=1212.819,-97.478,-37.842,179.398,5.426,149.129
C04404=1212.824,-97.728,-37.831,179.396,5.427,149.130
C04405=1212.829,-97.978,-37.821,179.394,5.426,149.131
C04406=1212.835,-98.227,-37.811,179.391,5.427,149.132
C04407=1212.840,-98.478,-37.800,179.389,5.426,149.132
C04408=1212.845,-98.727,-37.790,179.387,5.426,149.133
C04409=1212.850,-98.976,-37.780,179.384,5.426,149.133
C04410=1212.855,-99.227,-37.770,179.382,5.426,149.134
C04411=1212.861,-99.476,-37.759,179.380,5.426,149.135
C04412=1212.867,-99.726,-37.749,179.378,5.426,149.135
C04413=1212.872,-99.976,-37.739,179.375,5.425,149.136
C04414=1212.877,-100.226,-37.728,179.373,5.426,149.137
C04415=1212.881,-100.476,-37.718,179.371,5.425,149.137
C04416=1212.888,-100.746,-37.707,179.369,5.426,149.138
C04417=1212.893,-101.018,-37.696,179.366,5.425,149.139
C04418=1212.899,-101.289,-37.685,179.363,5.425,149.140
C04419=1212.905,-101.560,-37.674,179.361,5.425,149.140
C04420=1212.910,-101.810,-37.664,179.358,5.425,149.141
C04421=1212.915,-102.060,-37.653,179.356,5.425,149.142
C04422=1212.920,-102.310,-37.643,179.354,5.424,149.142
C04423=1212.925,-102.559,-37.633,179.352,5.425,149.143
C04424=1212.931,-102.809,-37.623,179.349,5.424,149.144
C04425=1212.936,-103.059,-37.612,179.347,5.425,149.144
C04426=1212.941,-103.309,-37.602,179.345,5.424,149.145
C04427=1212.947,-103.558,-37.592,179.343,5.424,149.146
C04428=1212.951,-103.808,-37.582,179.340,5.424,149.146
C04429=1212.957,-104.058,-37.572,179.338,5.424,149.147
C04430=1212.962,-104.307,-37.562,179.336,5.424,149.148
C04431=1212.967,-104.557,-37.551,179.334,5.424,149.148
C04432=1212.972,-104.807,-37.541,179.331,5.423,149.149
C04433=1212.978,-105.056,-37.531,179.329,5.424,149.150
C04434=1212.984,-105.306,-37.521,179.327,5.423,149.150
C04435=1212.989,-105.556,-37.510,179.324,5.424,149.151
C04436=1212.994,-105.806,-37.502,179.322,5.423,149.152
C04437=1212.999,-106.055,-37.491,179.320,5.423,149.152
C04438=1213.004,-106.306,-37.481,179.318,5.423,149.153
C04439=1213.009,-106.555,-37.471,179.315,5.423,149.154
C04440=1213.015,-106.804,-37.461,179.313,5.423,149.154
C04441=1213.020,-107.055,-37.450,179.311,5.423,149.155
C04442=1213.025,-107.304,-37.441,179.308,5.422,149.156
C04443=1213.031,-107.554,-37.431,179.306,5.423,149.156
C04444=1213.036,-107.804,-37.421,179.304,5.422,149.157
C04445=1213.041,-108.054,-37.410,179.302,5.423,149.158
C04446=1213.046,-108.303,-37.401,179.299,5.422,149.158
C04447=1213.052,-108.553,-37.391,179.297,5.422,149.159
C04448=1213.057,-108.802,-37.380,179.295,5.422,149.160
C04449=1213.062,-109.053,-37.371,179.293,5.422,149.160
C04450=1213.067,-109.302,-37.361,179.290,5.423,149.161
C04451=1213.073,-109.552,-37.351,179.288,5.422,149.162
C04452=1213.078,-109.801,-37.341,179.286,5.422,149.162
C04453=1213.083,-110.052,-37.331,179.284,5.422,149.163
C04454=1213.089,-110.301,-37.321,179.281,5.422,149.164
C04455=1213.094,-110.551,-37.311,179.279,5.421,149.164
C04456=1213.099,-110.800,-37.301,179.277,5.422,149.165
C04457=1213.104,-111.051,-37.292,179.274,5.421,149.166
C04458=1213.109,-111.300,-37.282,179.272,5.422,149.166
C04459=1213.115,-111.550,-37.272,179.270,5.421,149.167
C04460=1213.120,-111.799,-37.262,179.268,5.421,149.168
C04461=1213.125,-112.050,-37.252,179.265,5.421,149.168
C04462=1213.130,-112.299,-37.242,179.263,5.421,149.169
C04463=1213.136,-112.549,-37.232,179.261,5.421,149.170
C04464=1213.141,-112.799,-37.223,179.259,5.421,149.170
C04465=1213.146,-113.048,-37.213,179.256,5.420,149.171
C04466=1213.151,-113.298,-37.203,179.254,5.421,149.172
C04467=1213.156,-113.547,-37.193,179.252,5.420,149.172
C04468=1213.162,-113.798,-37.183,179.250,5.420,149.173
C04469=1213.168,-114.047,-37.173,179.247,5.420,149.174
C04470=1213.173,-114.297,-37.164,179.245,5.420,149.174
C04471=1213.178,-114.547,-37.154,179.243,5.420,149.175
C04472=1213.183,-114.797,-37.144,179.241,5.420,149.175
C04473=1213.189,-115.047,-37.135,179.239,5.420,149.176
C04474=1213.193,-115.296,-37.125,179.236,5.420,149.177
C04475=1213.199,-115.545,-37.115,179.234,5.420,149.178
C04476=1213.204,-115.795,-37.106,179.232,5.419,149.178
C04477=1213.209,-116.046,-37.095,179.230,5.420,149.179
C04478=1213.215,-116.295,-37.085,179.227,5.419,149.180
C04479=1213.220,-116.545,-37.076,179.225,5.420,149.180
C04480=1213.226,-116.795,-37.066,179.223,5.419,149.181
C04481=1213.231,-117.044,-37.057,179.221,5.419,149.181
C04482=1213.236,-117.294,-37.047,179.218,5.419,149.182
C04483=1213.242,-117.544,-37.038,179.216,5.419,149.183
C04484=1213.247,-117.794,-37.027,179.214,5.419,149.183
C04485=1213.251,-118.043,-37.018,179.212,5.419,149.184
C04486=1213.257,-118.293,-37.008,179.209,5.419,149.185
C04487=1213.262,-118.543,-36.999,179.207,5.419,149.185
C04488=1213.268,-118.793,-36.989,179.205,5.418,149.186
C04489=1213.273,-119.042,-36.980,179.203,5.419,149.187
C04490=1213.278,-119.292,-36.971,179.201,5.419,149.187
C04491=1213.283,-119.542,-36.960,179.198,5.419,149.188
C04492=1213.288,-119.792,-36.951,179.196,5.419,149.189
C04493=1213.294,-120.042,-36.941,179.194,5.418,149.189
C04494=1213.299,-120.291,-36.932,179.192,5.418,149.190
C04495=1213.305,-120.541,-36.922,179.189,5.418,149.191
C04496=1213.310,-120.791,-36.913,179.187,5.418,149.191
C04497=1213.315,-121.040,-36.903,179.185,5.418,149.192
C04498=1213.321,-121.290,-36.894,179.182,5.418,149.193
C04499=1213.325,-121.539,-36.884,179.180,5.417,149.193
C04500=1213.331,-121.790,-36.875,179.178,5.418,149.194
C04501=1213.336,-122.039,-36.865,179.176,5.417,149.195
C04502=1213.341,-122.290,-36.855,179.173,5.418,149.195
C04503=1213.346,-122.539,-36.846,179.172,5.418,149.196
C04504=1213.352,-122.789,-36.836,179.169,5.417,149.197
C04505=1213.357,-123.039,-36.827,179.167,5.418,149.197
C04506=1213.362,-123.288,-36.818,179.164,5.417,149.198
C04507=1213.368,-123.538,-36.808,179.163,5.417,149.198
C04508=1213.373,-123.788,-36.799,179.160,5.417,149.199
C04509=1213.378,-124.037,-36.790,179.158,5.417,149.200
C04510=1213.384,-124.288,-36.780,179.156,5.416,149.200
C04511=1213.389,-124.537,-36.771,179.154,5.417,149.201
C04512=1213.395,-124.787,-36.761,179.151,5.416,149.202
C04513=1213.400,-125.036,-36.752,179.149,5.417,149.203
C04514=1213.404,-125.287,-36.742,179.147,5.417,149.203
C04515=1213.410,-125.537,-36.733,179.145,5.416,149.204
C04516=1213.415,-125.786,-36.723,179.143,5.417,149.204
C04517=1213.420,-126.036,-36.714,179.140,5.416,149.205
C04518=1213.426,-126.286,-36.705,179.138,5.416,149.206
C04519=1213.431,-126.535,-36.695,179.136,5.416,149.206
C04520=1213.010,-126.546,-36.733,179.132,5.419,149.208
C04521=1213.004,-126.296,-36.742,179.134,5.420,149.208
C04522=1212.999,-126.047,-36.752,179.136,5.420,149.207
C04523=1212.994,-125.797,-36.761,179.139,5.420,149.206
C04524=1212.988,-125.547,-36.770,179.141,5.420,149.206
C04525=1212.983,-125.297,-36.780,179.143,5.420,149.205
C04526=1212.978,-125.048,-36.789,179.145,5.420,149.204
C04527=1212.972,-124.797,-36.798,179.147,5.420,149.204
C04528=1212.968,-124.548,-36.808,179.149,5.420,149.203
C04529=1212.962,-124.298,-36.817,179.151,5.420,149.202
C04530=1212.957,-124.049,-36.827,179.154,5.420,149.202
C04531=1212.952,-123.799,-36.836,179.156,5.420,149.201
C04532=1212.946,-123.549,-36.845,179.158,5.421,149.201
C04533=1212.941,-123.299,-36.855,179.160,5.420,149.200
C04534=1212.936,-123.050,-36.864,179.163,5.421,149.199
C04535=1212.930,-122.800,-36.874,179.165,5.421,149.199
C04536=1212.925,-122.550,-36.883,179.167,5.421,149.198
C04537=1212.920,-122.300,-36.893,179.169,5.421,149.197
C04538=1212.915,-122.050,-36.902,179.172,5.420,149.196
C04539=1212.910,-121.800,-36.911,179.174,5.421,149.196
C04540=1212.904,-121.551,-36.921,179.176,5.421,149.195
C04541=1212.899,-121.301,-36.930,179.179,5.421,149.195
C04542=1212.893,-121.051,-36.941,179.181,5.421,149.194
C04543=1212.888,-120.802,-36.949,179.183,5.422,149.193
C04544=1212.883,-120.552,-36.959,179.185,5.421,149.193
C04545=1212.877,-120.302,-36.969,179.188,5.422,149.192
C04546=1212.873,-120.052,-36.979,179.189,5.422,149.191
C04547=1212.867,-119.802,-36.988,179.192,5.422,149.191
C04548=1212.862,-119.553,-36.998,179.194,5.422,149.190
C04549=1212.856,-119.303,-37.007,179.197,5.422,149.189
C04550=1212.851,-119.053,-37.017,179.198,5.422,149.189
C04551=1212.846,-118.803,-37.026,179.201,5.422,149.188
C04552=1212.841,-118.554,-37.036,179.203,5.422,149.187
C04553=1212.835,-118.304,-37.045,179.205,5.422,149.187
C04554=1212.831,-118.054,-37.055,179.207,5.423,149.186
C04555=1212.825,-117.804,-37.065,179.209,5.422,149.185
C04556=1212.820,-117.554,-37.074,179.212,5.423,149.185
C04557=1212.814,-117.305,-37.085,179.214,5.422,149.184
C04558=1212.809,-117.055,-37.094,179.216,5.423,149.184
C04559=1212.803,-116.806,-37.104,179.218,5.423,149.183
C04560=1212.798,-116.556,-37.113,179.221,5.423,149.182
C04561=1212.793,-116.305,-37.123,179.223,5.423,149.181
C04562=1212.788,-116.056,-37.133,179.225,5.423,149.181
C04563=1212.782,-115.806,-37.142,179.227,5.423,149.180
C04564=1212.778,-115.557,-37.152,179.230,5.423,149.179
C04565=1212.772,-115.307,-37.161,179.232,5.423,149.179
C04566=1212.767,-115.057,-37.171,179.234,5.424,149.178
C04567=1212.762,-114.807,-37.182,179.237,5.423,149.178
C04568=1212.757,-114.557,-37.191,179.239,5.423,149.177
C04569=1212.751,-114.308,-37.201,179.241,5.423,149.176
C04570=1212.745,-114.058,-37.211,179.243,5.423,149.176
C04571=1212.740,-113.808,-37.220,179.246,5.424,149.175
C04572=1212.735,-113.559,-37.230,179.248,5.423,149.174
C04573=1212.730,-113.309,-37.240,179.250,5.424,149.173
C04574=1212.725,-113.059,-37.250,179.252,5.424,149.173
C04575=1212.720,-112.810,-37.259,179.255,5.424,149.172
C04576=1212.714,-112.560,-37.269,179.257,5.424,149.172
C04577=1212.708,-112.310,-37.279,179.259,5.424,149.171
C04578=1212.704,-112.060,-37.289,179.261,5.424,149.170
C04579=1212.698,-111.810,-37.299,179.264,5.425,149.170
C04580=1212.693,-111.561,-37.308,179.266,5.424,149.169
C04581=1212.688,-111.311,-37.318,179.268,5.425,149.168
C04582=1212.683,-111.061,-37.329,179.270,5.425,149.168
C04583=1212.678,-110.811,-37.338,179.273,5.425,149.167
C04584=1212.672,-110.561,-37.348,179.275,5.425,149.166
C04585=1212.666,-110.312,-37.358,179.277,5.425,149.166
C04586=1212.662,-110.062,-37.368,179.280,5.425,149.165
C04587=1212.656,-109.812,-37.378,179.282,5.426,149.164
C04588=1212.651,-109.562,-37.387,179.284,5.425,149.164
C04589=1212.646,-109.313,-37.397,179.287,5.426,149.163
C04590=1212.640,-109.063,-37.408,179.289,5.425,149.162
C04591=1212.636,-108.813,-37.417,179.291,5.426,149.162
C04592=1212.630,-108.564,-37.428,179.293,5.426,149.161
C04593=1212.624,-108.314,-37.437,179.295,5.425,149.160
C04594=1212.620,-108.064,-37.447,179.298,5.426,149.160
C04595=1212.614,-107.814,-37.457,179.299,5.426,149.159
C04596=1212.609,-107.565,-37.468,179.302,5.426,149.158
C04597=1212.603,-107.315,-37.478,179.304,5.426,149.158
C04598=1212.599,-107.065,-37.487,179.307,5.426,149.157
C04599=1212.593,-106.815,-37.497,179.309,5.426,149.156
C04600=1212.587,-106.566,-37.507,179.311,5.427,149.156
C04601=1212.583,-106.316,-37.517,179.313,5.426,149.155
C04602=1212.578,-106.066,-37.528,179.316,5.427,149.154
C04603=1212.572,-105.817,-37.538,179.318,5.426,149.154
C04604=1212.567,-105.567,-37.547,179.321,5.427,149.153
C04605=1212.562,-105.317,-37.558,179.322,5.427,149.152
C04606=1212.556,-105.067,-37.568,179.325,5.427,149.152
C04607=1212.551,-104.817,-37.578,179.327,5.427,149.151
C04608=1212.546,-104.567,-37.588,179.330,5.427,149.150
C04609=1212.541,-104.318,-37.598,179.331,5.427,149.150
C04610=1212.535,-104.068,-37.608,179.334,5.428,149.149
C04611=1212.530,-103.818,-37.619,179.336,5.427,149.148
C04612=1212.525,-103.569,-37.628,179.339,5.428,149.148
C04613=1212.520,-103.319,-37.639,179.341,5.427,149.147
C04614=1212.515,-103.069,-37.649,179.343,5.428,149.147
C04615=1212.509,-102.819,-37.659,179.345,5.428,149.146
C04616=1212.504,-102.570,-37.669,179.348,5.428,149.145
C04617=1212.499,-102.320,-37.680,179.350,5.428,149.144
C04618=1212.494,-102.070,-37.690,179.352,5.428,149.144
C04619=1212.488,-101.821,-37.700,179.354,5.428,149.143
C04620=1212.483,-101.571,-37.711,179.357,5.429,149.142
C04621=1212.477,-101.300,-37.721,179.359,5.428,149.142
C04622=1212.471,-101.028,-37.733,179.361,5.429,149.141
C04623=1212.466,-100.757,-37.744,179.364,5.429,149.140
C04624=1212.460,-100.487,-37.754,179.366,5.429,149.140
C04625=1212.455,-100.236,-37.765,179.369,5.429,149.139
C04626=1212.450,-99.987,-37.775,179.371,5.429,149.138
C04627=1212.445,-99.737,-37.786,179.374,5.429,149.137
C04628=1212.439,-99.487,-37.796,179.376,5.429,149.137
C04629=1212.434,-99.237,-37.806,179.378,5.430,149.136
C04630=1212.429,-98.988,-37.816,179.380,5.429,149.136
C04631=1212.424,-98.738,-37.826,179.383,5.430,149.135
C04632=1212.419,-98.488,-37.837,179.385,5.429,149.134
C04633=1212.413,-98.238,-37.847,179.387,5.430,149.133
C04634=1212.408,-97.989,-37.857,179.389,5.430,149.133
C04635=1212.403,-97.738,-37.868,179.392,5.430,149.132
C04636=1212.397,-97.489,-37.878,179.394,5.430,149.132
C04637=1212.392,-97.239,-37.888,179.397,5.430,149.131
C04638=1212.387,-96.990,-37.899,179.399,5.430,149.130
C04639=1212.382,-96.740,-37.909,179.401,5.430,149.129
C04640=1212.377,-96.490,-37.920,179.403,5.430,149.129
C04641=1212.371,-96.241,-37.930,179.406,5.431,149.128
C04642=1212.366,-95.990,-37.940,179.408,5.430,149.127
C04643=1212.361,-95.741,-37.951,179.410,5.431,149.127
C04644=1212.355,-95.491,-37.961,179.412,5.430,149.126
C04645=1212.350,-95.242,-37.972,179.415,5.431,149.126
C04646=1212.345,-94.992,-37.982,179.417,5.431,149.125
C04647=1212.340,-94.742,-37.993,179.419,5.431,149.124
C04648=1212.334,-94.492,-38.003,179.422,5.432,149.123
C04649=1212.329,-94.242,-38.014,179.424,5.431,149.123
C04650=1212.323,-93.993,-38.024,179.427,5.432,149.122
C04651=1212.319,-93.743,-38.035,179.428,5.432,149.122
C04652=1212.314,-93.494,-38.045,179.431,5.432,149.121
C04653=1212.308,-93.244,-38.055,179.433,5.432,149.120
C04654=1212.303,-92.994,-38.066,179.436,5.432,149.119
C04655=1212.298,-92.744,-38.076,179.438,5.432,149.119
C04656=1212.293,-92.495,-38.087,179.441,5.432,149.118
C04657=1212.287,-92.245,-38.097,179.442,5.432,149.117
C04658=1212.282,-91.995,-38.108,179.445,5.433,149.117
C04659=1212.277,-91.745,-38.118,179.447,5.432,149.116
C04660=1212.272,-91.496,-38.129,179.450,5.433,149.115
C04661=1212.267,-91.246,-38.140,179.452,5.432,149.115
C04662=1212.262,-90.996,-38.150,179.454,5.433,149.114
C04663=1212.256,-90.747,-38.161,179.456,5.433,149.113
C04664=1212.251,-90.497,-38.172,179.459,5.433,149.113
C04665=1212.246,-90.247,-38.182,179.461,5.433,149.112
C04666=1212.241,-89.997,-38.192,179.463,5.433,149.111
C04667=1212.235,-89.748,-38.203,179.466,5.433,149.111
C04668=1212.230,-89.498,-38.214,179.468,5.433,149.110
C04669=1212.224,-89.248,-38.225,179.470,5.433,149.109
C04670=1212.219,-88.998,-38.236,179.472,5.434,149.109
C04671=1212.214,-88.749,-38.246,179.475,5.434,149.108
C04672=1212.209,-88.499,-38.257,179.477,5.434,149.107
C04673=1212.203,-88.250,-38.268,179.480,5.434,149.107
C04674=1212.198,-87.999,-38.278,179.482,5.434,149.106
C04675=1212.193,-87.750,-38.288,179.484,5.435,149.105
C04676=1212.188,-87.500,-38.300,179.486,5.434,149.105
C04677=1212.183,-87.251,-38.310,179.489,5.435,149.104
C04678=1212.178,-87.001,-38.321,179.491,5.434,149.103
C04679=1212.173,-86.751,-38.332,179.494,5.435,149.103
C04680=1212.167,-86.501,-38.342,179.496,5.434,149.102
C04681=1212.163,-86.252,-38.353,179.498,5.435,149.101
C04682=1212.156,-86.002,-38.364,179.500,5.435,149.101
C04683=1212.152,-85.752,-38.375,179.503,5.435,149.100
C04684=1212.146,-85.503,-38.386,179.505,5.435,149.099
C04685=1212.141,-85.252,-38.396,179.507,5.435,149.098
C04686=1212.136,-85.003,-38.407,179.510,5.436,149.098
C04687=1212.131,-84.753,-38.418,179.512,5.435,149.097
C04688=1212.126,-84.504,-38.429,179.514,5.436,149.097
C04689=1212.120,-84.254,-38.439,179.517,5.436,149.096
C04690=1212.115,-84.004,-38.451,179.519,5.436,149.095
C04691=1212.109,-83.755,-38.461,179.521,5.436,149.094
C04692=1212.105,-83.505,-38.473,179.524,5.436,149.094
C04693=1212.100,-83.255,-38.483,179.526,5.436,149.093
C04694=1212.094,-83.006,-38.494,179.528,5.437,149.093
C04695=1212.089,-82.756,-38.505,179.530,5.437,149.092
C04696=1212.084,-82.507,-38.516,179.533,5.437,149.091
C04697=1212.078,-82.256,-38.527,179.535,5.437,149.090
C04698=1212.074,-82.007,-38.538,179.538,5.437,149.090
C04699=1212.068,-81.757,-38.548,179.540,5.437,149.089
C04700=1212.063,-81.507,-38.560,179.542,5.437,149.088
C04701=1212.058,-81.258,-38.570,179.545,5.438,149.088
C04702=1212.052,-81.008,-38.582,179.547,5.438,149.087
C04703=1212.047,-80.758,-38.592,179.549,5.438,149.086
C04704=1212.042,-80.509,-38.603,179.552,5.438,149.086
C04705=1212.037,-80.259,-38.614,179.554,5.438,149.085
C04706=1212.032,-80.009,-38.626,179.556,5.438,149.084
C04707=1212.026,-79.760,-38.637,179.559,5.438,149.084
C04708=1212.021,-79.509,-38.647,179.561,5.439,149.083
C04709=1212.017,-79.260,-38.658,179.563,5.439,149.082
C04710=1212.011,-79.010,-38.669,179.566,5.439,149.082
C04711=1212.006,-78.760,-38.680,179.568,5.439,149.081
C04712=1212.001,-78.511,-38.692,179.571,5.439,149.080
C04713=1211.995,-78.261,-38.702,179.573,5.439,149.080
C04714=1211.990,-78.011,-38.714,179.575,5.439,149.079
C04715=1211.985,-77.762,-38.725,179.577,5.439,149.078
C04716=1211.980,-77.512,-38.735,179.580,5.440,149.078
C04717=1211.975,-77.262,-38.747,179.582,5.440,149.077
C04718=1211.970,-77.012,-38.759,179.584,5.440,149.076
C04719=1211.964,-76.763,-38.769,179.587,5.440,149.076
C04720=1211.959,-76.513,-38.780,179.589,5.440,149.075
C04721=1211.954,-76.263,-38.792,179.592,5.440,149.074
C04722=1211.948,-76.014,-38.802,179.594,5.440,149.073
C04723=1211.943,-75.764,-38.813,179.596,5.441,149.073
C04724=1211.938,-75.514,-38.825,179.598,5.440,149.072
C04725=1211.933,-75.244,-38.837,179.601,5.441,149.071
C04726=1211.927,-74.973,-38.849,179.604,5.441,149.071
C04727=1211.921,-74.702,-38.861,179.607,5.441,149.070
C04728=1211.915,-74.432,-38.873,179.609,5.441,149.069
C04729=1211.910,-74.182,-38.884,179.611,5.441,149.068
C04730=1211.906,-73.933,-38.896,179.613,5.441,149.068
C04731=1211.899,-73.683,-38.906,179.616,5.442,149.067
C04732=1211.895,-73.433,-38.918,179.618,5.441,149.067
C04733=1211.889,-73.183,-38.930,179.621,5.442,149.066
C04734=1211.884,-72.934,-38.940,179.623,5.442,149.065
C04735=1211.879,-72.685,-38.952,179.625,5.442,149.064
C04736=1211.874,-72.434,-38.963,179.628,5.442,149.064
C04737=1211.869,-72.185,-38.974,179.630,5.442,149.063
C04738=1211.863,-71.935,-38.986,179.632,5.443,149.063
C04739=1211.858,-71.686,-38.997,179.634,5.443,149.062
C04740=1211.853,-71.436,-39.008,179.637,5.443,149.061
C04741=1211.848,-71.186,-39.019,179.640,5.443,149.060
C04742=1211.842,-70.937,-39.030,179.642,5.443,149.060
C04743=1211.837,-70.687,-39.042,179.644,5.444,149.059
C04744=1211.832,-70.437,-39.054,179.646,5.443,149.058
C04745=1211.828,-70.187,-39.065,179.649,5.444,149.058
C04746=1211.822,-69.938,-39.076,179.651,5.443,149.057
C04747=1211.817,-69.688,-39.087,179.653,5.444,149.056
C04748=1211.811,-69.438,-39.099,179.656,5.445,149.056
C04749=1211.806,-69.188,-39.110,179.658,5.444,149.055
C04750=1211.801,-68.938,-39.122,179.661,5.445,149.054
C04751=1211.796,-68.690,-39.133,179.663,5.444,149.054
C04752=1211.790,-68.440,-39.145,179.666,5.445,149.053
C04753=1211.786,-68.190,-39.156,179.668,5.445,149.052
C04754=1211.780,-67.940,-39.168,179.670,5.445,149.051
C04755=1211.776,-67.690,-39.179,179.673,5.446,149.051
C04756=1211.769,-67.441,-39.191,179.675,5.445,149.050
C04757=1211.764,-67.191,-39.201,179.677,5.446,149.050
C04758=1211.760,-66.941,-39.213,179.679,5.445,149.049
C04759=1211.754,-66.691,-39.225,179.682,5.446,149.048
C04760=1211.750,-66.442,-39.236,179.685,5.446,149.047
C04761=1211.744,-66.193,-39.247,179.687,5.446,149.047
C04762=1211.738,-65.943,-39.259,179.689,5.446,149.046
C04763=1211.734,-65.693,-39.271,179.692,5.446,149.045
C04764=1211.728,-65.443,-39.282,179.694,5.447,149.045
C04765=1211.723,-65.193,-39.294,179.696,5.447,149.044
C04766=1211.718,-64.943,-39.306,179.698,5.447,149.043
C04767=1211.713,-64.695,-39.317,179.701,5.447,149.043
C04768=1211.707,-64.445,-39.328,179.703,5.447,149.042
C04769=1211.703,-64.195,-39.340,179.706,5.448,149.041
C04770=1211.697,-63.945,-39.352,179.709,5.448,149.041
C04771=1211.692,-63.695,-39.363,179.711,5.448,149.040
C04772=1211.687,-63.445,-39.375,179.713,5.448,149.039
C04773=1211.682,-63.196,-39.386,179.715,5.448,149.039
C04774=1211.676,-62.947,-39.398,179.718,5.449,149.038
C04775=1211.671,-62.697,-39.410,179.720,5.449,149.037
C04776=1211.666,-62.448,-39.421,179.722,5.449,149.037
C04777=1211.661,-62.198,-39.433,179.725,5.449,149.036
C04778=1211.656,-61.948,-39.445,179.727,5.449,149.035
C04779=1211.651,-61.698,-39.457,179.730,5.449,149.034
C04780=1211.645,-61.448,-39.468,179.732,5.450,149.034
C04781=1211.641,-61.199,-39.480,179.735,5.449,149.033
C04782=1211.635,-60.949,-39.491,179.737,5.450,149.033
C04783=1211.630,-60.700,-39.503,179.739,5.450,149.032
C04784=1211.625,-60.450,-39.514,179.741,5.450,149.031
C04785=1211.620,-60.200,-39.527,179.744,5.451,149.030
C04786=1211.615,-59.951,-39.538,179.746,5.450,149.030
C04787=1211.609,-59.701,-39.550,179.749,5.451,149.029
C04788=1211.604,-59.451,-39.562,179.751,5.450,149.028
C04789=1211.599,-59.201,-39.573,179.754,5.451,149.028
C04790=1211.594,-58.951,-39.585,179.756,5.451,149.027
C04791=1211.589,-58.702,-39.598,179.758,5.451,149.026
C04792=1211.584,-58.452,-39.609,179.761,5.452,149.026
C04793=1211.579,-58.203,-39.621,179.763,5.452,149.025
C04794=1211.573,-57.953,-39.633,179.765,5.452,149.024
C04795=1211.568,-57.704,-39.644,179.768,5.452,149.024
C04796=1211.563,-57.454,-39.656,179.770,5.452,149.023
C04797=1211.557,-57.204,-39.668,179.773,5.453,149.022
C04798=1211.553,-56.955,-39.680,179.775,5.452,149.022
C04799=1211.547,-56.705,-39.691,179.777,5.453,149.021
C04800=1211.542,-56.456,-39.704,179.780,5.453,149.020
C04801=1211.537,-56.206,-39.715,179.782,5.453,149.020
C04802=1211.532,-55.956,-39.727,179.784,5.454,149.019
C04803=1211.527,-55.706,-39.739,179.787,5.454,149.018
C04804=1211.522,-55.457,-39.751,179.789,5.454,149.018
C04805=1211.517,-55.207,-39.763,179.792,5.454,149.017
C04806=1211.511,-54.957,-39.775,179.794,5.454,149.016
C04807=1211.506,-54.707,-39.787,179.797,5.454,149.015
C04808=1211.501,-54.458,-39.799,179.799,5.455,149.015
C04809=1211.496,-54.208,-39.811,179.801,5.454,149.014
C04810=1211.491,-53.958,-39.823,179.804,5.455,149.013
C04811=1211.485,-53.709,-39.835,179.807,5.455,149.013
C04812=1211.481,-53.459,-39.846,179.808,5.455,149.012
C04813=1211.475,-53.209,-39.858,179.811,5.456,149.011
C04814=1211.470,-52.960,-39.871,179.813,5.455,149.011
C04815=1211.465,-52.710,-39.883,179.816,5.456,149.010
C04816=1211.460,-52.461,-39.894,179.818,5.456,149.009
C04817=1211.455,-52.211,-39.907,179.820,5.456,149.009
C04818=1211.450,-51.961,-39.919,179.823,5.456,149.008
C04819=1211.444,-51.712,-39.931,179.826,5.457,149.007
C04820=1211.439,-51.462,-39.943,179.828,5.457,149.006
C04821=1211.434,-51.212,-39.955,179.830,5.457,149.006
C04822=1211.429,-50.963,-39.967,179.832,5.457,149.005
C04823=1211.424,-50.713,-39.979,179.835,5.458,149.005
C04824=1211.419,-50.464,-39.991,179.837,5.458,149.004
C04825=1211.413,-50.214,-40.003,179.839,5.458,149.003
C04826=1211.408,-49.964,-40.015,179.842,5.458,149.002
C04827=1211.403,-49.714,-40.028,179.845,5.459,149.002
C04828=1211.399,-49.464,-40.040,179.847,5.458,149.001
C04829=1211.392,-49.195,-40.053,179.850,5.459,149.000
C04830=1211.387,-48.925,-40.066,179.852,5.459,149.000
C04831=1211.381,-48.655,-40.079,179.855,5.460,148.999
C04832=1211.376,-48.385,-40.092,179.857,5.459,148.998
C04833=1211.371,-48.135,-40.105,179.860,5.460,148.998
C04834=1211.365,-47.885,-40.116,179.862,5.460,148.997
C04835=1211.360,-47.636,-40.129,179.864,5.460,148.996
C04836=1211.355,-47.386,-40.141,179.867,5.460,148.995
C04837=1211.350,-47.136,-40.154,179.870,5.461,148.995
C04838=1211.346,-46.887,-40.166,179.872,5.460,148.994
C04839=1211.340,-46.637,-40.178,179.875,5.461,148.993
C04840=1211.335,-46.388,-40.190,179.877,5.461,148.993
C04841=1211.330,-46.138,-40.202,179.879,5.461,148.992
C04842=1211.325,-45.889,-40.215,179.882,5.462,148.991
C04843=1211.319,-45.639,-40.227,179.883,5.462,148.991
C04844=1211.314,-45.389,-40.239,179.886,5.462,148.990
C04845=1211.309,-45.139,-40.251,179.889,5.463,148.989
C04846=1211.303,-44.890,-40.264,179.891,5.462,148.989
C04847=1211.299,-44.640,-40.277,179.894,5.463,148.988
C04848=1211.294,-44.390,-40.289,179.896,5.463,148.987
C04849=1211.288,-44.141,-40.301,179.898,5.463,148.987
C04850=1211.283,-43.891,-40.313,179.901,5.463,148.986
C04851=1211.278,-43.642,-40.326,179.904,5.464,148.985
C04852=1211.273,-43.392,-40.338,179.906,5.463,148.984
C04853=1211.267,-43.142,-40.350,179.908,5.464,148.984
C04854=1211.263,-42.892,-40.363,179.911,5.465,148.983
C04855=1211.258,-42.643,-40.376,179.913,5.464,148.983
C04856=1211.252,-42.393,-40.388,179.915,5.465,148.982
C04857=1211.247,-42.144,-40.400,179.918,5.465,148.981
C04858=1211.242,-41.894,-40.412,179.920,5.465,148.980
C04859=1211.237,-41.644,-40.425,179.923,5.465,148.980
C04860=1211.231,-41.395,-40.437,179.925,5.466,148.979
C04861=1211.227,-41.145,-40.450,179.927,5.466,148.978
C04862=1211.221,-40.895,-40.462,179.930,5.466,148.978
C04863=1211.216,-40.646,-40.475,179.933,5.466,148.977
C04864=1211.211,-40.397,-40.487,179.935,5.466,148.976
C04865=1211.206,-40.147,-40.499,179.937,5.467,148.976
C04866=1211.201,-39.897,-40.512,179.940,5.467,148.975
C04867=1211.196,-39.647,-40.525,179.942,5.467,148.974
C04868=1211.191,-39.398,-40.538,179.944,5.468,148.974
C04869=1211.186,-39.148,-40.549,179.947,5.468,148.973
C04870=1211.180,-38.899,-40.562,179.949,5.468,148.972
C04871=1211.176,-38.649,-40.575,179.952,5.468,148.972
C04872=1211.171,-38.399,-40.588,179.955,5.469,148.971
C04873=1211.165,-38.149,-40.600,179.957,5.468,148.970
C04874=1211.160,-37.900,-40.613,179.959,5.469,148.970
C04875=1211.154,-37.651,-40.625,179.962,5.469,148.969
C04876=1211.150,-37.401,-40.638,179.964,5.469,148.968
C04877=1211.145,-37.151,-40.651,179.966,5.470,148.968
C04878=1211.139,-36.901,-40.663,179.969,5.470,148.967
C04879=1211.134,-36.652,-40.675,179.971,5.470,148.966
C04880=1211.129,-36.403,-40.688,179.974,5.470,148.966
C04881=1211.124,-36.152,-40.701,179.976,5.471,148.965
C04882=1211.119,-35.903,-40.714,179.978,5.471,148.964
C04883=1211.114,-35.654,-40.727,179.981,5.471,148.963
C04884=1211.108,-35.404,-40.739,179.984,5.471,148.963
C04885=1211.104,-35.154,-40.752,179.986,5.472,148.962
C04886=1211.098,-34.904,-40.764,179.988,5.472,148.961
C04887=1211.093,-34.655,-40.777,179.991,5.472,148.961
C04888=1211.088,-34.405,-40.790,179.993,5.473,148.960
C04889=1211.083,-34.155,-40.803,179.995,5.473,148.959
C04890=1211.078,-33.906,-40.815,179.998,5.473,148.959
C04891=1211.073,-33.657,-40.828,-179.999,5.474,148.958
C04892=1211.068,-33.407,-40.841,-179.997,5.473,148.957
C04893=1211.062,-33.157,-40.854,-179.995,5.474,148.957
C04894=1211.057,-32.907,-40.866,-179.992,5.474,148.956
C04895=1211.052,-32.658,-40.879,-179.990,5.474,148.955
C04896=1211.047,-32.408,-40.892,-179.987,5.474,148.955
C04897=1211.042,-32.159,-40.904,-179.985,5.475,148.954
C04898=1211.036,-31.909,-40.917,-179.982,5.475,148.953
C04899=1211.032,-31.659,-40.930,-179.980,5.475,148.952
C04900=1211.027,-31.410,-40.943,-179.978,5.476,148.952
C04901=1211.022,-31.160,-40.956,-179.975,5.476,148.951
C04902=1211.016,-30.910,-40.969,-179.973,5.476,148.951
C04903=1211.011,-30.661,-40.982,-179.970,5.476,148.950
C04904=1211.006,-30.411,-40.994,-179.968,5.477,148.949
C04905=1211.001,-30.161,-41.007,-179.965,5.477,148.949
C04906=1210.996,-29.912,-41.021,-179.963,5.477,148.948
C04907=1210.991,-29.662,-41.033,-179.960,5.478,148.947
C04908=1210.986,-29.412,-41.046,-179.957,5.478,148.946
C04909=1210.981,-29.163,-41.059,-179.955,5.478,148.946
C04910=1210.975,-28.914,-41.073,-179.953,5.478,148.945
C04911=1210.971,-28.664,-41.086,-179.951,5.479,148.945
C04912=1210.966,-28.415,-41.098,-179.949,5.479,148.944
C04913=1210.960,-28.165,-41.111,-179.946,5.479,148.943
C04914=1210.955,-27.915,-41.124,-179.943,5.480,148.942
C04915=1210.950,-27.666,-41.137,-179.941,5.480,148.942
C04916=1210.944,-27.416,-41.150,-179.938,5.480,148.941
C04917=1210.940,-27.166,-41.163,-179.936,5.480,148.940
C04918=1210.935,-26.917,-41.176,-179.933,5.481,148.940
C04919=1210.929,-26.667,-41.189,-179.931,5.480,148.939
C04920=1210.925,-26.418,-41.203,-179.928,5.481,148.938
C04921=1210.919,-26.168,-41.215,-179.926,5.481,148.938
C04922=1210.914,-25.918,-41.229,-179.923,5.482,148.937
C04923=1210.909,-25.669,-41.241,-179.921,5.482,148.936
C04924=1210.904,-25.419,-41.254,-179.919,5.482,148.936
C04925=1210.899,-25.169,-41.268,-179.916,5.483,148.935
C04926=1210.894,-24.920,-41.280,-179.914,5.483,148.934
C04927=1210.889,-24.670,-41.294,-179.911,5.483,148.934
C04928=1210.883,-24.421,-41.307,-179.909,5.484,148.933
C04929=1210.878,-24.171,-41.320,-179.906,5.484,148.932
C04930=1210.873,-23.921,-41.333,-179.904,5.484,148.932
C04931=1210.868,-23.672,-41.346,-179.901,5.484,148.931
C04932=1210.864,-23.422,-41.359,-179.899,5.485,148.930
C04933=1210.857,-23.153,-41.373,-179.896,5.485,148.929
C04934=1210.852,-22.884,-41.388,-179.893,5.486,148.929
C04935=1210.847,-22.614,-41.402,-179.891,5.485,148.928
C04936=1210.841,-22.344,-41.416,-179.889,5.486,148.927
C04937=1210.836,-22.095,-41.430,-179.886,5.486,148.927
C04938=1210.831,-21.846,-41.443,-179.883,5.487,148.926
C04939=1210.826,-21.596,-41.456,-179.881,5.486,148.925
C04940=1210.820,-21.346,-41.469,-179.879,5.487,148.925
C04941=1210.816,-21.096,-41.483,-179.876,5.487,148.924
C04942=1210.810,-20.847,-41.496,-179.873,5.488,148.923
C04943=1210.806,-20.597,-41.509,-179.871,5.488,148.923
C04944=1210.801,-20.348,-41.522,-179.869,5.488,148.922
C04945=1210.795,-20.098,-41.536,-179.866,5.489,148.921
C04946=1210.790,-19.848,-41.548,-179.864,5.489,148.921
C04947=1210.785,-19.599,-41.563,-179.862,5.489,148.920
C04948=1210.780,-19.349,-41.575,-179.859,5.490,148.919
C04949=1210.774,-19.100,-41.588,-179.856,5.490,148.919
C04950=1210.770,-18.850,-41.602,-179.854,5.491,148.918
C04951=1210.764,-18.601,-41.615,-179.852,5.490,148.917
C04952=1210.759,-18.350,-41.629,-179.849,5.491,148.917
C04953=1210.754,-18.102,-41.642,-179.846,5.491,148.916
C04954=1210.749,-17.851,-41.656,-179.844,5.492,148.915
C04955=1210.744,-17.603,-41.669,-179.842,5.491,148.914
C04956=1210.739,-17.352,-41.683,-179.839,5.492,148.914
C04957=1210.734,-17.103,-41.695,-179.837,5.493,148.913
C04958=1210.729,-16.853,-41.709,-179.834,5.493,148.913
C04959=1210.724,-16.603,-41.722,-179.832,5.493,148.912
C04960=1210.719,-16.354,-41.736,-179.829,5.493,148.911
C04961=1210.714,-16.104,-41.749,-179.827,5.494,148.910
C04962=1210.709,-15.855,-41.763,-179.824,5.494,148.910
C04963=1210.703,-15.605,-41.777,-179.822,5.494,148.909
C04964=1210.699,-15.356,-41.790,-179.819,5.495,148.908
C04965=1210.693,-15.106,-41.804,-179.817,5.495,148.908
C04966=1210.689,-14.857,-41.817,-179.814,5.496,148.907
C04967=1210.683,-14.607,-41.831,-179.812,5.496,148.907
C04968=1210.678,-14.358,-41.844,-179.810,5.496,148.906
C04969=1210.673,-14.108,-41.857,-179.807,5.497,148.905
C04970=1210.668,-13.859,-41.871,-179.804,5.497,148.904
C04971=1210.663,-13.609,-41.884,-179.802,5.497,148.904
C04972=1210.658,-13.359,-41.899,-179.800,5.497,148.903
C04973=1210.652,-13.110,-41.912,-179.797,5.498,148.902
C04974=1210.648,-12.860,-41.925,-179.794,5.498,148.902
C04975=1210.642,-12.611,-41.939,-179.792,5.499,148.901
C04976=1210.637,-12.361,-41.953,-179.790,5.498,148.900
C04977=1210.632,-12.111,-41.966,-179.787,5.499,148.900
C04978=1210.627,-11.862,-41.980,-179.785,5.500,148.899
C04979=1210.622,-11.612,-41.994,-179.782,5.500,148.898
C04980=1210.617,-11.363,-42.007,-179.780,5.500,148.898
C04981=1210.612,-11.113,-42.021,-179.777,5.500,148.897
C04982=1210.606,-10.863,-42.034,-179.775,5.501,148.896
C04983=1210.602,-10.614,-42.048,-179.772,5.501,148.896
C04984=1210.597,-10.364,-42.062,-179.769,5.502,148.895
C04985=1210.591,-10.115,-42.075,-179.767,5.502,148.894
C04986=1210.587,-9.865,-42.089,-179.765,5.502,148.894
C04987=1210.582,-9.616,-42.103,-179.762,5.503,148.893
C04988=1210.576,-9.366,-42.116,-179.760,5.504,148.892
C04989=1210.572,-9.117,-42.130,-179.758,5.503,148.892
C04990=1210.566,-8.868,-42.144,-179.755,5.504,148.891
C04991=1210.561,-8.617,-42.158,-179.752,5.504,148.890
C04992=1210.556,-8.367,-42.172,-179.750,5.505,148.890
C04993=1210.551,-8.119,-42.185,-179.747,5.505,148.889
C04994=1210.546,-7.868,-42.199,-179.745,5.505,148.888
C04995=1210.541,-7.619,-42.213,-179.742,5.505,148.888
C04996=1210.536,-7.370,-42.227,-179.740,5.506,148.887
C04997=1210.531,-7.120,-42.241,-179.737,5.506,148.886
C04998=1210.526,-6.870,-42.254,-179.735,5.507,148.886
C04999=1210.521,-6.621,-42.268,-179.733,5.507,148.885
C05000=1210.516,-6.371,-42.282,-179.730,5.507,148.884
C05001=1210.511,-6.122,-42.296,-179.728,5.508,148.884
C05002=1210.506,-5.872,-42.309,-179.725,5.508,148.883
C05003=1210.501,-5.623,-42.324,-179.722,5.509,148.882
C05004=1210.496,-5.373,-42.338,-179.720,5.509,148.882
C05005=1210.490,-5.124,-42.352,-179.718,5.509,148.881
C05006=1210.485,-4.873,-42.365,-179.715,5.510,148.880
C05007=1210.481,-4.624,-42.379,-179.712,5.510,148.880
C05008=1210.476,-4.374,-42.393,-179.710,5.511,148.879
C05009=1210.470,-4.125,-42.407,-179.708,5.511,148.878
C05010=1210.465,-3.876,-42.421,-179.705,5.511,148.878
C05011=1210.460,-3.626,-42.436,-179.703,5.512,148.877
C05012=1210.454,-3.376,-42.449,-179.700,5.512,148.876
C05013=1210.450,-3.127,-42.463,-179.697,5.513,148.876
C05014=1210.445,-2.877,-42.477,-179.695,5.512,148.875
C05015=1210.440,-2.628,-42.491,-179.693,5.513,148.874
C05016=1210.435,-2.379,-42.505,-179.690,5.513,148.874
C05017=1210.430,-2.129,-42.519,-179.688,5.514,148.873
C05018=1210.425,-1.879,-42.534,-179.685,5.515,148.872
C05019=1210.419,-1.630,-42.548,-179.683,5.514,148.872
C05020=1210.415,-1.380,-42.561,-179.680,5.515,148.871
C05021=1210.410,-1.130,-42.575,-179.678,5.515,148.870
C05022=1210.405,-0.881,-42.589,-179.675,5.516,148.870
C05023=1210.399,-0.632,-42.603,-179.672,5.516,148.869
C05024=1210.394,-0.382,-42.617,-179.670,5.516,148.868
C05025=1210.389,-0.132,-42.632,-179.668,5.517,148.868
C05026=1210.384,0.118,-42.646,-179.665,5.517,148.867
C05027=1210.379,0.367,-42.660,-179.663,5.518,148.866
C05028=1210.374,0.616,-42.674,-179.660,5.519,148.866
C05029=1210.369,0.866,-42.688,-179.658,5.519,148.865
C05030=1210.364,1.116,-42.703,-179.656,5.519,148.864
C05031=1210.359,1.365,-42.717,-179.653,5.519,148.864
C05032=1210.353,1.614,-42.731,-179.650,5.520,148.863
C05033=1210.348,1.864,-42.745,-179.648,5.520,148.862
C05034=1210.344,2.114,-42.759,-179.645,5.521,148.862
C05035=1210.339,2.364,-42.774,-179.642,5.521,148.861
C05036=1210.334,2.613,-42.788,-179.641,5.521,148.861
C05037=1210.328,2.882,-42.802,-179.638,5.521,148.860
C05038=1210.322,3.151,-42.818,-179.635,5.522,148.859
C05039=1210.317,3.420,-42.834,-179.632,5.522,148.858
C05040=1210.312,3.689,-42.849,-179.630,5.523,148.858
C05041=1210.307,3.939,-42.863,-179.627,5.523,148.857
C05042=1210.302,4.188,-42.877,-179.624,5.524,148.856
C05043=1210.296,4.437,-42.891,-179.622,5.524,148.855
C05044=1210.291,4.687,-42.906,-179.619,5.525,148.855
C05045=1210.287,4.937,-42.920,-179.617,5.526,148.854
C05046=1210.282,5.186,-42.935,-179.615,5.526,148.854
C05047=1210.277,5.436,-42.949,-179.612,5.526,148.853
C05048=1210.272,5.685,-42.963,-179.609,5.527,148.852
C05049=1210.266,5.934,-42.977,-179.607,5.527,148.852
C05050=1210.261,6.184,-42.992,-179.604,5.528,148.851
C05051=1210.256,6.434,-43.006,-179.601,5.528,148.850
C05052=1210.252,6.683,-43.020,-179.600,5.528,148.850
C05053=1210.246,6.933,-43.036,-179.597,5.529,148.849
C05054=1210.241,7.183,-43.050,-179.595,5.529,148.848
C05055=1210.236,7.432,-43.064,-179.592,5.530,148.848
C05056=1210.231,7.682,-43.079,-179.589,5.530,148.847
C05057=1210.226,7.931,-43.093,-179.587,5.531,148.846
C05058=1210.221,8.180,-43.108,-179.584,5.531,148.846
C05059=1210.216,8.430,-43.122,-179.582,5.531,148.845
C05060=1210.211,8.679,-43.136,-179.579,5.531,148.844
C05061=1210.206,8.929,-43.150,-179.577,5.532,148.844
C05062=1210.202,9.178,-43.165,-179.574,5.533,148.843
C05063=1210.196,9.428,-43.180,-179.572,5.533,148.842
C05064=1210.191,9.678,-43.194,-179.569,5.534,148.842
C05065=1210.186,9.928,-43.209,-179.566,5.534,148.841
C05066=1210.181,10.176,-43.223,-179.564,5.534,148.840
C05067=1210.176,10.426,-43.238,-179.562,5.535,148.840
C05068=1210.171,10.676,-43.252,-179.559,5.535,148.839
C05069=1210.165,10.926,-43.267,-179.557,5.536,148.839
C05070=1210.160,11.175,-43.282,-179.554,5.536,148.838
C05071=1210.156,11.424,-43.296,-179.552,5.537,148.837
C05072=1210.151,11.674,-43.310,-179.549,5.538,148.836
C05073=1210.146,11.923,-43.325,-179.546,5.538,148.836
C05074=1210.141,12.173,-43.340,-179.544,5.538,148.835
C05075=1210.135,12.423,-43.355,-179.542,5.538,148.834
C05076=1210.131,12.672,-43.370,-179.539,5.539,148.834
C05077=1210.126,12.922,-43.384,-179.537,5.540,148.833
C05078=1210.121,13.171,-43.399,-179.534,5.540,148.833
C05079=1210.115,13.421,-43.414,-179.532,5.541,148.832
C05080=1210.110,13.671,-43.428,-179.529,5.541,148.831
C05081=1210.106,13.920,-43.443,-179.526,5.542,148.831
C05082=1210.101,14.169,-43.457,-179.524,5.541,148.830
C05083=1210.095,14.419,-43.473,-179.522,5.542,148.829
C05084=1210.090,14.668,-43.487,-179.519,5.543,148.829
C05085=1210.085,14.918,-43.501,-179.517,5.543,148.828
C05086=1210.081,15.167,-43.516,-179.514,5.544,148.827
C05087=1210.075,15.417,-43.531,-179.511,5.544,148.827
C05088=1210.070,15.666,-43.546,-179.509,5.545,148.826
C05089=1210.066,15.916,-43.560,-179.506,5.545,148.825
C05090=1210.061,16.165,-43.575,-179.504,5.545,148.825
C05091=1210.055,16.415,-43.590,-179.501,5.546,148.824
C05092=1210.051,16.664,-43.605,-179.499,5.547,148.823
C05093=1210.046,16.914,-43.620,-179.497,5.547,148.823
C05094=1210.040,17.163,-43.635,-179.494,5.548,148.822
C05095=1210.035,17.413,-43.649,-179.491,5.548,148.821
C05096=1210.031,17.662,-43.664,-179.489,5.549,148.821
C05097=1210.025,17.912,-43.679,-179.486,5.549,148.820
C05098=1210.020,18.161,-43.694,-179.483,5.550,148.819
C05099=1210.015,18.411,-43.709,-179.481,5.551,148.819
C05100=1210.010,18.660,-43.724,-179.479,5.550,148.818
C05101=1210.005,18.910,-43.738,-179.476,5.551,148.818
C05102=1210.000,19.159,-43.753,-179.474,5.551,148.817
C05103=1209.995,19.409,-43.769,-179.471,5.552,148.816
C05104=1209.990,19.658,-43.783,-179.469,5.552,148.816
C05105=1209.985,19.907,-43.798,-179.466,5.553,148.815
C05106=1209.980,20.157,-43.813,-179.464,5.554,148.814
C05107=1209.975,20.407,-43.828,-179.461,5.554,148.814
C05108=1209.970,20.656,-43.844,-179.458,5.555,148.813
C05109=1209.965,20.906,-43.858,-179.456,5.555,148.812
C05110=1209.960,21.155,-43.873,-179.453,5.556,148.812
C05111=1209.954,21.405,-43.888,-179.451,5.555,148.811
C05112=1209.950,21.655,-43.903,-179.448,5.556,148.810
C05113=1209.945,21.904,-43.919,-179.446,5.557,148.810
C05114=1209.940,22.154,-43.933,-179.444,5.557,148.809
C05115=1209.934,22.403,-43.949,-179.441,5.558,148.808
C05116=1209.930,22.652,-43.964,-179.438,5.558,148.808
C05117=1209.925,22.902,-43.978,-179.436,5.559,148.807
C05118=1209.920,23.151,-43.994,-179.433,5.560,148.806
C05119=1209.915,23.400,-44.009,-179.431,5.560,148.806
C05120=1209.909,23.650,-44.024,-179.428,5.561,148.805
C05121=1209.905,23.899,-44.038,-179.426,5.561,148.805
C05122=1209.900,24.150,-44.054,-179.423,5.562,148.804
C05123=1209.895,24.399,-44.069,-179.420,5.562,148.803
C05124=1209.890,24.648,-44.085,-179.418,5.562,148.803
C05125=1209.885,24.898,-44.099,-179.416,5.563,148.802
C05126=1209.879,25.147,-44.115,-179.413,5.564,148.801
C05127=1209.875,25.396,-44.130,-179.411,5.564,148.801
C05128=1209.869,25.646,-44.145,-179.408,5.565,148.800
C05129=1209.865,25.896,-44.160,-179.405,5.565,148.799
C05130=1209.860,26.145,-44.176,-179.403,5.566,148.799
C05131=1209.855,26.395,-44.191,-179.400,5.566,148.798
C05132=1209.850,26.644,-44.206,-179.398,5.567,148.798
C05133=1209.845,26.893,-44.221,-179.395,5.568,148.797
C05134=1209.839,27.143,-44.236,-179.393,5.568,148.796
C05135=1209.835,27.393,-44.251,-179.390,5.569,148.796
C05136=1209.830,27.642,-44.267,-179.387,5.569,148.795
C05137=1209.824,27.892,-44.283,-179.385,5.570,148.794
C05138=1209.820,28.141,-44.298,-179.383,5.571,148.794
C05139=1209.814,28.390,-44.313,-179.380,5.571,148.793
C05140=1209.810,28.640,-44.329,-179.378,5.571,148.792
C05141=1209.804,28.909,-44.345,-179.375,5.572,148.792
C05142=1209.799,29.178,-44.362,-179.372,5.573,148.791
C05143=1209.794,29.446,-44.378,-179.369,5.573,148.790
C05144=1209.788,29.715,-44.395,-179.367,5.574,148.790
C05145=1209.784,29.964,-44.410,-179.364,5.574,148.789
C05146=1209.778,30.213,-44.425,-179.362,5.575,148.788
C05147=1209.773,30.463,-44.441,-179.359,5.575,148.788
C05148=1209.769,30.713,-44.456,-179.356,5.576,148.787
C05149=1209.763,30.962,-44.472,-179.354,5.576,148.786
C05150=1209.758,31.211,-44.487,-179.351,5.577,148.786
C05151=1209.753,31.460,-44.502,-179.349,5.578,148.785
C05152=1209.749,31.711,-44.518,-179.346,5.578,148.785
C05153=1209.743,31.961,-44.533,-179.343,5.579,148.784
C05154=1209.738,32.210,-44.548,-179.341,5.579,148.783
C05155=1209.733,32.458,-44.564,-179.339,5.580,148.783
C05156=1209.728,32.709,-44.580,-179.337,5.580,148.782
C05157=1209.724,32.958,-44.595,-179.334,5.581,148.781
C05158=1209.718,33.207,-44.611,-179.331,5.581,148.781
C05159=1209.713,33.456,-44.627,-179.329,5.582,148.780
C05160=1209.709,33.706,-44.642,-179.326,5.582,148.779
C05161=1209.703,33.956,-44.658,-179.324,5.583,148.779
C05162=1209.698,34.205,-44.673,-179.321,5.584,148.778
C05163=1209.694,34.455,-44.688,-179.319,5.584,148.778
C05164=1209.689,34.704,-44.704,-179.316,5.585,148.777
C05165=1209.683,34.954,-44.720,-179.313,5.585,148.776
C05166=1209.678,35.203,-44.735,-179.311,5.586,148.776
C05167=1209.674,35.453,-44.751,-179.309,5.587,148.775
C05168=1209.668,35.702,-44.766,-179.306,5.587,148.774
C05169=1209.663,35.952,-44.782,-179.303,5.588,148.774
C05170=1209.659,36.201,-44.798,-179.301,5.588,148.773
C05171=1209.654,36.450,-44.813,-179.298,5.589,148.772
C05172=1209.649,36.700,-44.829,-179.296,5.590,148.772
C05173=1209.644,36.950,-44.845,-179.293,5.590,148.771
C05174=1209.638,37.199,-44.861,-179.291,5.591,148.771
C05175=1209.634,37.448,-44.876,-179.288,5.591,148.770
C05176=1209.629,37.698,-44.892,-179.285,5.592,148.769
C05177=1209.624,37.947,-44.908,-179.283,5.593,148.769
C05178=1209.618,38.196,-44.923,-179.280,5.593,148.768
C05179=1209.614,38.447,-44.939,-179.278,5.594,148.767
C05180=1209.609,38.696,-44.954,-179.275,5.594,148.767
C05181=1209.604,38.944,-44.971,-179.273,5.595,148.766
C05182=1209.599,39.195,-44.987,-179.270,5.595,148.765
C05183=1209.594,39.444,-45.002,-179.268,5.596,148.765
C05184=1209.588,39.693,-45.018,-179.265,5.597,148.764
C05185=1209.584,39.943,-45.034,-179.262,5.597,148.764
C05186=1209.578,40.192,-45.050,-179.260,5.598,148.763
C05187=1209.574,40.441,-45.065,-179.257,5.599,148.762
C05188=1209.569,40.691,-45.081,-179.255,5.599,148.762
C05189=1209.564,40.940,-45.097,-179.252,5.600,148.761
C05190=1209.559,41.190,-45.113,-179.250,5.600,148.760
C05191=1209.554,41.440,-45.129,-179.247,5.601,148.760
C05192=1209.549,41.689,-45.145,-179.244,5.602,148.759
C05193=1209.544,41.939,-45.161,-179.242,5.602,148.759
C05194=1209.539,42.188,-45.177,-179.240,5.603,148.758
C05195=1209.534,42.436,-45.192,-179.237,5.604,148.757
C05196=1209.529,42.687,-45.208,-179.234,5.604,148.757
C05197=1209.524,42.936,-45.224,-179.232,5.605,148.756
C05198=1209.520,43.185,-45.241,-179.230,5.606,148.756
C05199=1209.514,43.435,-45.256,-179.227,5.606,148.755
C05200=1209.509,43.685,-45.272,-179.224,5.607,148.754
C05201=1209.504,43.934,-45.288,-179.222,5.607,148.754
C05202=1209.499,44.183,-45.304,-179.220,5.608,148.753
C05203=1209.494,44.433,-45.321,-179.217,5.609,148.752
C05204=1209.489,44.682,-45.336,-179.214,5.609,148.752
C05205=1209.485,44.932,-45.353,-179.212,5.610,148.751
C05206=1209.479,45.181,-45.369,-179.209,5.610,148.750
C05207=1209.474,45.431,-45.384,-179.207,5.611,148.750
C05208=1209.469,45.680,-45.401,-179.204,5.612,148.749
C05209=1209.465,45.930,-45.417,-179.202,5.612,148.749
C05210=1209.459,46.179,-45.433,-179.199,5.613,148.748
C05211=1209.454,46.428,-45.449,-179.196,5.613,148.747
C05212=1209.450,46.678,-45.465,-179.194,5.615,148.747
C05213=1209.444,46.927,-45.481,-179.191,5.616,148.746
C05214=1209.440,47.176,-45.498,-179.188,5.616,148.746
C05215=1209.434,47.426,-45.513,-179.186,5.617,148.745
C05216=1209.430,47.675,-45.530,-179.183,5.618,148.744
C05217=1209.424,47.925,-45.545,-179.181,5.618,148.744
C05218=1209.420,48.174,-45.562,-179.178,5.619,148.743
C05219=1209.415,48.424,-45.578,-179.176,5.619,148.742
C05220=1209.410,48.673,-45.594,-179.173,5.620,148.742
C05221=1209.405,48.922,-45.611,-179.171,5.621,148.741
C05222=1209.400,49.172,-45.627,-179.168,5.621,148.741
C05223=1209.395,49.421,-45.643,-179.166,5.622,148.740
C05224=1209.390,49.671,-45.659,-179.163,5.622,148.739
C05225=1209.385,49.920,-45.675,-179.161,5.623,148.739
C05226=1209.381,50.169,-45.692,-179.158,5.624,148.738
C05227=1209.376,50.419,-45.708,-179.155,5.624,148.737
C05228=1209.370,50.668,-45.725,-179.153,5.625,148.737
C05229=1209.365,50.918,-45.741,-179.150,5.625,148.736
C05230=1209.360,51.167,-45.757,-179.148,5.626,148.736
C05231=1209.356,51.417,-45.774,-179.145,5.627,148.735
C05232=1209.350,51.666,-45.789,-179.143,5.627,148.734
C05233=1209.346,51.916,-45.806,-179.140,5.629,148.734
C05234=1209.341,52.164,-45.822,-179.137,5.630,148.733
C05235=1209.336,52.415,-45.838,-179.135,5.630,148.733
C05236=1209.330,52.664,-45.855,-179.132,5.631,148.732
C05237=1209.326,52.913,-45.872,-179.130,5.631,148.731
C05238=1209.321,53.163,-45.888,-179.127,5.632,148.731
C05239=1209.316,53.412,-45.904,-179.125,5.633,148.730
C05240=1209.311,53.661,-45.921,-179.122,5.633,148.729
C05241=1209.306,53.910,-45.937,-179.119,5.634,148.729
C05242=1209.301,54.161,-45.953,-179.117,5.635,148.728
C05243=1209.296,54.410,-45.970,-179.115,5.635,148.728
C05244=1209.291,54.659,-45.986,-179.112,5.636,148.727
C05245=1209.287,54.927,-46.005,-179.109,5.637,148.726
C05246=1209.281,55.196,-46.022,-179.106,5.638,148.726
C05247=1209.275,55.464,-46.040,-179.104,5.638,148.725
C05248=1209.270,55.733,-46.057,-179.101,5.639,148.724
C05249=1209.265,55.982,-46.074,-179.098,5.639,148.724
C05250=1209.261,56.232,-46.090,-179.096,5.640,148.723
C05251=1209.255,56.481,-46.107,-179.093,5.642,148.723
C05252=1209.250,56.730,-46.124,-179.090,5.642,148.722
C05253=1209.246,56.980,-46.140,-179.088,5.643,148.721
C05254=1209.241,57.230,-46.156,-179.086,5.644,148.721
C05255=1209.235,57.479,-46.173,-179.083,5.644,148.720
C05256=1209.231,57.728,-46.190,-179.080,5.645,148.720
C05257=1209.226,57.977,-46.206,-179.078,5.645,148.719
C05258=1209.220,58.227,-46.224,-179.075,5.646,148.718
C05259=1209.216,58.476,-46.240,-179.073,5.647,148.718
C05260=1209.211,58.725,-46.257,-179.070,5.647,148.717
C05261=1209.206,58.975,-46.273,-179.068,5.648,148.716
C05262=1209.201,59.224,-46.290,-179.065,5.650,148.716
C05263=1209.196,59.474,-46.306,-179.062,5.650,148.715
C05264=1209.191,59.723,-46.323,-179.060,5.651,148.715
C05265=1209.186,59.973,-46.340,-179.057,5.652,148.714
C05266=1209.181,60.222,-46.356,-179.055,5.652,148.714
C05267=1209.177,60.471,-46.373,-179.052,5.653,148.713
C05268=1209.171,60.721,-46.390,-179.050,5.653,148.712
C05269=1209.167,60.971,-46.407,-179.047,5.654,148.712
C05270=1209.162,61.219,-46.423,-179.045,5.655,148.711
C05271=1209.157,61.469,-46.440,-179.042,5.656,148.710
C05272=1209.152,61.719,-46.457,-179.039,5.657,148.710
C05273=1209.146,61.968,-46.474,-179.037,5.658,148.709
C05274=1209.142,62.217,-46.491,-179.034,5.658,148.709
C05275=1209.137,62.467,-46.507,-179.032,5.659,148.708
C05276=1209.131,62.716,-46.524,-179.029,5.659,148.707
C05277=1209.127,62.965,-46.541,-179.027,5.660,148.707
C05278=1209.122,63.215,-46.558,-179.024,5.661,148.706
C05279=1209.118,63.464,-46.576,-179.021,5.661,148.706
C05280=1209.113,63.713,-46.592,-179.019,5.663,148.705
C05281=1209.107,63.963,-46.609,-179.016,5.664,148.705
C05282=1209.103,64.212,-46.626,-179.013,5.664,148.704
C05283=1209.098,64.462,-46.643,-179.011,5.665,148.703
C05284=1209.093,64.711,-46.659,-179.009,5.666,148.703
C05285=1209.087,64.960,-46.677,-179.006,5.666,148.702
C05286=1209.083,65.210,-46.693,-179.003,5.667,148.701
C05287=1209.078,65.459,-46.710,-179.001,5.668,148.701
C05288=1209.073,65.708,-46.728,-178.998,5.669,148.700
C05289=1209.068,65.957,-46.744,-178.995,5.670,148.700
C05290=1209.063,66.207,-46.762,-178.993,5.670,148.699
C05291=1209.059,66.457,-46.778,-178.991,5.671,148.699
C05292=1209.053,66.706,-46.795,-178.988,5.672,148.698
C05293=1209.048,66.955,-46.812,-178.985,5.672,148.697
C05294=1209.043,67.204,-46.830,-178.983,5.673,148.697
C05295=1209.039,67.454,-46.846,-178.980,5.675,148.696
C05296=1209.034,67.704,-46.864,-178.977,5.675,148.696
C05297=1209.029,67.953,-46.880,-178.975,5.676,148.695
C05298=1209.024,68.202,-46.898,-178.973,5.677,148.694
C05299=1209.019,68.451,-46.915,-178.970,5.677,148.694
C05300=1209.014,68.701,-46.932,-178.967,5.678,148.693
C05301=1209.010,68.950,-46.949,-178.965,5.679,148.693
C05302=1209.005,69.200,-46.967,-178.962,5.680,148.692
C05303=1208.999,69.449,-46.984,-178.959,5.681,148.691
C05304=1208.994,69.698,-47.000,-178.957,5.681,148.691
C05305=1208.989,69.947,-47.018,-178.955,5.682,148.690
C05306=1208.985,70.197,-47.035,-178.952,5.683,148.690
C05307=1208.980,70.447,-47.052,-178.949,5.683,148.689
C05308=1208.975,70.696,-47.069,-178.947,5.685,148.688
C05309=1208.970,70.945,-47.087,-178.944,5.685,148.688
C05310=1208.965,71.195,-47.104,-178.941,5.686,148.687
C05311=1208.960,71.443,-47.121,-178.939,5.687,148.687
C05312=1208.955,71.693,-47.138,-178.937,5.687,148.686
C05313=1208.951,71.943,-47.155,-178.934,5.688,148.685
C05314=1208.946,72.192,-47.173,-178.931,5.690,148.685
C05315=1208.941,72.442,-47.190,-178.929,5.690,148.684
C05316=1208.936,72.691,-47.207,-178.926,5.691,148.684
C05317=1208.931,72.940,-47.225,-178.923,5.691,148.683
C05318=1208.926,73.190,-47.242,-178.921,5.692,148.683
C05319=1208.921,73.438,-47.259,-178.919,5.693,148.682
C05320=1208.916,73.688,-47.276,-178.915,5.694,148.681
C05321=1208.911,73.937,-47.294,-178.913,5.695,148.681
C05322=1208.907,74.187,-47.311,-178.911,5.696,148.680
C05323=1208.901,74.436,-47.328,-178.908,5.696,148.680
C05324=1208.896,74.686,-47.346,-178.906,5.697,148.679
C05325=1208.892,74.935,-47.363,-178.903,5.699,148.678
C05326=1208.887,75.184,-47.381,-178.900,5.699,148.678
C05327=1208.882,75.434,-47.398,-178.898,5.700,148.677
C05328=1208.878,75.683,-47.416,-178.895,5.701,148.677
C05329=1208.872,75.933,-47.433,-178.893,5.701,148.676
C05330=1208.867,76.182,-47.451,-178.891,5.702,148.676
C05331=1208.862,76.431,-47.468,-178.887,5.704,148.675
C05332=1208.857,76.680,-47.485,-178.885,5.704,148.674
C05333=1208.853,76.929,-47.503,-178.883,5.705,148.674
C05334=1208.847,77.179,-47.520,-178.880,5.706,148.673
C05335=1208.842,77.428,-47.538,-178.877,5.706,148.673
C05336=1208.838,77.677,-47.555,-178.875,5.708,148.672
C05337=1208.833,77.927,-47.573,-178.872,5.709,148.671
C05338=1208.828,78.176,-47.590,-178.869,5.709,148.671
C05339=1208.823,78.426,-47.608,-178.867,5.710,148.670
C05340=1208.818,78.675,-47.626,-178.865,5.711,148.670
C05341=1208.814,78.924,-47.643,-178.861,5.712,148.669
C05342=1208.809,79.173,-47.661,-178.859,5.713,148.669
C05343=1208.804,79.423,-47.679,-178.857,5.714,148.668
C05344=1208.798,79.672,-47.696,-178.854,5.714,148.667
C05345=1208.794,79.922,-47.714,-178.852,5.715,148.667
C05346=1208.789,80.170,-47.731,-178.849,5.716,148.666
C05347=1208.784,80.420,-47.749,-178.846,5.717,148.666
C05348=1208.779,80.669,-47.767,-178.844,5.718,148.665
C05349=1208.774,80.938,-47.785,-178.841,5.719,148.665
C05350=1208.769,81.207,-47.805,-178.838,5.720,148.664
C05351=1208.764,81.475,-47.824,-178.836,5.720,148.663
C05352=1208.758,81.744,-47.843,-178.832,5.722,148.663
C05353=1208.753,81.993,-47.861,-178.830,5.723,148.662
C05354=1208.749,82.242,-47.879,-178.828,5.723,148.662
C05355=1208.744,82.491,-47.897,-178.825,5.724,148.661
C05356=1208.739,82.741,-47.913,-178.822,5.726,148.660
C05357=1208.734,82.990,-47.931,-178.820,5.726,148.660
C05358=1208.729,83.239,-47.949,-178.817,5.727,148.659
C05359=1208.724,83.488,-47.967,-178.815,5.728,148.659
C05360=1208.719,83.738,-47.985,-178.812,5.729,148.658
C05361=1208.714,83.987,-48.003,-178.810,5.730,148.658
C05362=1208.709,84.236,-48.021,-178.807,5.731,148.657
C05363=1208.704,84.486,-48.039,-178.804,5.731,148.656
C05364=1208.700,84.735,-48.057,-178.802,5.732,148.656
C05365=1208.695,84.984,-48.075,-178.799,5.734,148.655
C05366=1208.689,85.234,-48.092,-178.796,5.734,148.655
C05367=1208.684,85.483,-48.110,-178.794,5.735,148.654
C05368=1208.680,85.733,-48.128,-178.792,5.736,148.654
C05369=1208.675,85.982,-48.146,-178.788,5.737,148.653
C05370=1208.670,86.231,-48.164,-178.786,5.738,148.652
C05371=1208.666,86.480,-48.181,-178.784,5.739,148.652
C05372=1208.661,86.729,-48.199,-178.781,5.739,148.651
C05373=1208.656,86.978,-48.217,-178.778,5.741,148.651
C05374=1208.651,87.227,-48.235,-178.776,5.741,148.650
C05375=1208.647,87.477,-48.253,-178.774,5.742,148.650
C05376=1208.641,87.726,-48.271,-178.771,5.743,148.649
C05377=1208.636,87.977,-48.290,-178.768,5.744,148.648
C05378=1208.631,88.226,-48.308,-178.766,5.745,148.648
C05379=1208.626,88.475,-48.326,-178.763,5.746,148.647
C05380=1208.622,88.724,-48.344,-178.761,5.747,148.647
C05381=1208.617,88.973,-48.362,-178.758,5.748,148.646
C05382=1208.612,89.223,-48.380,-178.755,5.749,148.646
C05383=1208.607,89.472,-48.397,-178.753,5.750,148.645
C05384=1208.602,89.722,-48.416,-178.750,5.751,148.645
C05385=1208.598,89.971,-48.434,-178.748,5.752,148.644
C05386=1208.593,90.220,-48.452,-178.745,5.753,148.643
C05387=1208.588,90.469,-48.470,-178.742,5.753,148.643
C05388=1208.583,90.718,-48.488,-178.740,5.755,148.642
C05389=1208.578,90.967,-48.506,-178.737,5.755,148.642
C05390=1208.574,91.217,-48.525,-178.735,5.756,148.641
C05391=1208.568,91.466,-48.543,-178.732,5.757,148.641
C05392=1208.563,91.715,-48.561,-178.729,5.758,148.640
C05393=1208.558,91.965,-48.579,-178.727,5.759,148.640
C05394=1208.554,92.214,-48.597,-178.724,5.760,148.639
C05395=1208.549,92.464,-48.616,-178.722,5.762,148.639
C05396=1208.544,92.713,-48.634,-178.719,5.762,148.638
C05397=1208.539,92.962,-48.652,-178.716,5.763,148.637
C05398=1208.535,93.210,-48.670,-178.714,5.764,148.637
C05399=1208.529,93.460,-48.689,-178.711,5.765,148.636
C05400=1208.525,93.710,-48.707,-178.709,5.766,148.636
C05401=1208.520,93.959,-48.725,-178.706,5.767,148.635
C05402=1208.515,94.208,-48.743,-178.703,5.768,148.634
C05403=1208.510,94.457,-48.761,-178.701,5.769,148.634
C05404=1208.505,94.707,-48.781,-178.698,5.770,148.633
C05405=1208.500,94.956,-48.799,-178.696,5.771,148.633
C05406=1208.496,95.205,-48.817,-178.693,5.772,148.632
C05407=1208.491,95.454,-48.835,-178.690,5.773,148.632
C05408=1208.486,95.704,-48.853,-178.688,5.773,148.631
C05409=1208.481,95.953,-48.872,-178.685,5.775,148.631
C05410=1208.476,96.202,-48.890,-178.683,5.776,148.630
C05411=1208.471,96.452,-48.908,-178.680,5.776,148.630
C05412=1208.467,96.701,-48.927,-178.677,5.778,148.629
C05413=1208.461,96.950,-48.946,-178.675,5.779,148.628
C05414=1208.457,97.199,-48.964,-178.672,5.779,148.628
C05415=1208.452,97.449,-48.982,-178.670,5.780,148.627
C05416=1208.448,97.698,-49.001,-178.667,5.782,148.627
C05417=1208.442,97.947,-49.020,-178.665,5.783,148.626
C05418=1208.437,98.197,-49.038,-178.662,5.783,148.626
C05419=1208.433,98.446,-49.057,-178.659,5.785,148.625
C05420=1208.428,98.695,-49.075,-178.657,5.786,148.625
C05421=1208.423,98.945,-49.093,-178.654,5.786,148.624
C05422=1208.419,99.194,-49.112,-178.652,5.788,148.624
C05423=1208.414,99.443,-49.130,-178.649,5.788,148.623
C05424=1208.408,99.692,-49.150,-178.647,5.789,148.623
C05425=1208.404,99.942,-49.168,-178.644,5.791,148.622
C05426=1208.399,100.191,-49.186,-178.642,5.792,148.621
C05427=1208.394,100.440,-49.205,-178.639,5.792,148.621
C05428=1208.389,100.690,-49.223,-178.636,5.794,148.620
C05429=1208.385,100.938,-49.242,-178.634,5.795,148.620
C05430=1208.379,101.188,-49.261,-178.631,5.795,148.619
C05431=1208.375,101.437,-49.280,-178.628,5.797,148.619
C05432=1208.369,101.686,-49.298,-178.626,5.798,148.618
C05433=1208.365,101.936,-49.316,-178.624,5.799,148.618
C05434=1208.361,102.185,-49.335,-178.620,5.800,148.617
C05435=1208.355,102.434,-49.354,-178.618,5.801,148.617
C05436=1208.351,102.684,-49.373,-178.616,5.801,148.616
C05437=1208.346,102.933,-49.391,-178.612,5.803,148.615
C05438=1208.341,103.182,-49.410,-178.610,5.804,148.615
C05439=1208.336,103.431,-49.429,-178.608,5.804,148.614
C05440=1208.331,103.680,-49.448,-178.605,5.806,148.614
C05441=1208.326,103.929,-49.467,-178.602,5.807,148.613
C05442=1208.321,104.179,-49.486,-178.600,5.808,148.613
C05443=1208.317,104.428,-49.504,-178.597,5.809,148.612
C05444=1208.312,104.678,-49.523,-178.595,5.810,148.612
C05445=1208.307,104.926,-49.542,-178.592,5.811,148.611
C05446=1208.302,105.176,-49.560,-178.590,5.812,148.611
C05447=1208.297,105.425,-49.580,-178.587,5.813,148.610
C05448=1208.293,105.674,-49.598,-178.584,5.814,148.609
C05449=1208.288,105.924,-49.617,-178.582,5.815,148.609
C05450=1208.283,106.172,-49.636,-178.579,5.816,148.608
C05451=1208.278,106.422,-49.656,-178.576,5.818,148.608
C05452=1208.273,106.671,-49.674,-178.574,5.818,148.607
C05453=1208.268,106.939,-49.694,-178.571,5.820,148.607
C05454=1208.263,107.208,-49.715,-178.568,5.821,148.606
C05455=1208.257,107.476,-49.735,-178.565,5.822,148.606
C05456=1208.253,107.745,-49.755,-178.563,5.823,148.605
C05457=1208.247,107.994,-49.774,-178.560,5.824,148.605
C05458=1208.243,108.243,-49.793,-178.557,5.825,148.604
C05459=1208.238,108.492,-49.813,-178.555,5.826,148.604
C05460=1208.234,108.742,-49.831,-178.552,5.827,148.603
C05461=1208.228,108.991,-49.850,-178.550,5.828,148.602
C05462=1208.224,109.241,-49.870,-178.547,5.829,148.602
C05463=1208.219,109.490,-49.888,-178.545,5.831,148.601
C05464=1208.214,109.739,-49.908,-178.542,5.831,148.601
C05465=1208.209,109.988,-49.926,-178.539,5.833,148.600
C05466=1208.205,110.237,-49.946,-178.537,5.834,148.600
C05467=1208.199,110.486,-49.965,-178.535,5.835,148.599
C05468=1208.195,110.736,-49.984,-178.531,5.836,148.599
C05469=1208.190,110.985,-50.003,-178.529,5.837,148.598
C05470=1208.186,111.234,-50.022,-178.526,5.838,148.598
C05471=1208.180,111.483,-50.041,-178.524,5.839,148.597
C05472=1208.176,111.733,-50.061,-178.521,5.840,148.597
C05473=1208.171,111.981,-50.080,-178.519,5.842,148.596
C05474=1208.166,112.232,-50.099,-178.516,5.842,148.596
C05475=1208.161,112.480,-50.118,-178.513,5.844,148.595
C05476=1208.157,112.730,-50.137,-178.511,5.845,148.595
C05477=1208.151,112.979,-50.156,-178.509,5.846,148.594
C05478=1208.146,113.228,-50.176,-178.505,5.847,148.593
C05479=1208.142,113.477,-50.195,-178.503,5.848,148.593
C05480=1208.137,113.726,-50.214,-178.500,5.849,148.592
C05481=1208.132,113.975,-50.234,-178.498,5.850,148.592
C05482=1208.128,114.224,-50.253,-178.495,5.851,148.591
C05483=1208.123,114.474,-50.272,-178.493,5.853,148.591
C05484=1208.118,114.723,-50.292,-178.490,5.853,148.590
C05485=1208.113,114.973,-50.311,-178.487,5.855,148.590
C05486=1208.108,115.222,-50.329,-178.485,5.856,148.589
